LIN {X 0,Y 283.836,Z 555.722,A -85,B 0,C 180,E1 20309.781,E2 20309.781} C_VEL
LIN {X 0,Y 281.486,Z 550.799,A -85,B 0,C 180,E1 20310.705,E2 20310.705} C_VEL
LIN {X 0,Y 279.401,Z 540.674,A -85,B 0,C 180,E1 20314.395,E2 20314.395} C_VEL
LIN {X 0,Y 277.114,Z 531.716,A -85,B 0,C 180,E1 20318.183,E2 20318.183} C_VEL
LIN {X 0,Y 274.511,Z 522.89,A -85,B 0,C 180,E1 20322.608,E2 20322.608} C_VEL
LIN {X 0,Y 272.161,Z 516.128,A -85,B 0,C 180,E1 20326.833,E2 20326.833} C_VEL
LIN {X 0,Y 270.651,Z 512.243,A -85,B 0,C 180,E1 20329.786,E2 20329.786} C_VEL
LIN {X 0,Y 269.541,Z 509.144,A -85,B 0,C 180,E1 20332.54,E2 20332.54} C_VEL
LIN {X 0,Y 268.278,Z 505.702,A -85,B 0,C 180,E1 20336.367,E2 20336.367} C_VEL
LIN {X 0,Y 267.046,Z 502.186,A -85,B 0,C 180,E1 20343.219,E2 20343.219} C_VEL
LIN {X 0,Y 266.89,Z 501.903,A -85,B 0,C 180,E1 20348.618,E2 20348.618} C_VEL
LIN {X 0,Y 267.553,Z 502.917,A -85,B 0,C 180,E1 20352.744,E2 20352.744} C_VEL
LIN {X 0,Y 269.686,Z 507.312,A -85,B 0,C 180,E1 20359.492,E2 20359.492} C_VEL
LIN {X 0,Y 271.699,Z 511.865,A -85,B 0,C 180,E1 20363.648,E2 20363.648} C_VEL
LIN {X 0,Y 273.683,Z 516.523,A -85,B 0,C 180,E1 20366.949,E2 20366.949} C_VEL
LIN {X 0,Y 276.357,Z 522.601,A -85,B 0,C 180,E1 20370.562,E2 20370.562} C_VEL
LIN {X 0,Y 279.81,Z 531.752,A -85,B 0,C 180,E1 20374.871,E2 20374.871} C_VEL
LIN {X 0,Y 283.199,Z 541.616,A -85,B 0,C 180,E1 20378.676,E2 20378.676} C_VEL
LIN {X 0,Y 284.32,Z 544.973,A -85,B 0,C 180,E1 20379.794,E2 20379.794} C_VEL
LIN {X 0,Y 291.359,Z 556.974,A -85,B 0,C 180,E1 20382.037,E2 20382.037} C_VEL
LIN {X 0,Y 293.853,Z 561.883,A -85,B 0,C 180,E1 20382.784,E2 20382.784} C_VEL
LIN {X 0,Y 295.222,Z 584.167,A -85,B 0,C 180,E1 20383.897,E2 20383.897} C_VEL
LIN {X 0,Y 287.499,Z 725.367,A -85,B 0,C 180,E1 20387.325,E2 20387.325} C_VEL
LIN {X 0,Y 285.33,Z 743.573,A -85,B 0,C 180,E1 20388.063,E2 20388.063} C_VEL
LIN {X 0,Y 282.159,Z 761.285,A -85,B 0,C 180,E1 20389.11,E2 20389.11} C_VEL
LIN {X 0,Y 278.499,Z 777.354,A -85,B 0,C 180,E1 20390.413,E2 20390.413} C_VEL
LIN {X 0,Y 274.274,Z 793.21,A -85,B 0,C 180,E1 20392.102,E2 20392.102} C_VEL
LIN {X 0,Y 269.76,Z 808.181,A -85,B 0,C 180,E1 20394.153,E2 20394.153} C_VEL
LIN {X 0,Y 264.96,Z 822.734,A -85,B 0,C 180,E1 20396.698,E2 20396.698} C_VEL
LIN {X 0,Y 260.466,Z 835.727,A -85,B 0,C 180,E1 20399.555,E2 20399.555} C_VEL
LIN {X 0,Y 256.384,Z 847.663,A -85,B 0,C 180,E1 20402.853,E2 20402.853} C_VEL
LIN {X 0,Y 253.012,Z 858.122,A -85,B 0,C 180,E1 20406.476,E2 20406.476} C_VEL
LIN {X 0,Y 250.58,Z 867.042,A -85,B 0,C 180,E1 20410.417,E2 20410.417} C_VEL
LIN {X 0,Y 249.191,Z 874.327,A -85,B 0,C 180,E1 20414.644,E2 20414.644} C_VEL
LIN {X 0,Y 248.918,Z 879.669,A -85,B 0,C 180,E1 20418.884,E2 20418.884} C_VEL
LIN {X 0,Y 249.44,Z 883.153,A -85,B 0,C 180,E1 20423.094,E2 20423.094} C_VEL
LIN {X 0,Y 250.202,Z 884.696,A -85,B 0,C 180,E1 20426.793,E2 20426.793} C_VEL
LIN {X 0,Y 250.573,Z 884.807,A -85,B 0,C 180,E1 20430,E2 20430} C_VEL
LIN {X 0,Y 250.353,Z 883.594,A -85,B 0,C 180,E1 20433.206,E2 20433.206} C_VEL
LIN {X 0,Y 249.71,Z 880.685,A -85,B 0,C 180,E1 20436.9,E2 20436.9} C_VEL
LIN {X 0,Y 249.251,Z 876.121,A -85,B 0,C 180,E1 20440.641,E2 20440.641} C_VEL
LIN {X 0,Y 249.336,Z 869.417,A -85,B 0,C 180,E1 20444.634,E2 20444.634} C_VEL
LIN {X 0,Y 250.208,Z 861.167,A -85,B 0,C 180,E1 20448.403,E2 20448.403} C_VEL
LIN {X 0,Y 251.809,Z 851.451,A -85,B 0,C 180,E1 20451.916,E2 20451.916} C_VEL
LIN {X 0,Y 254.087,Z 840.281,A -85,B 0,C 180,E1 20455.168,E2 20455.168} C_VEL
LIN {X 0,Y 256.938,Z 827.315,A -85,B 0,C 180,E1 20458.217,E2 20458.217} C_VEL
LIN {X 0,Y 260.267,Z 812.638,A -85,B 0,C 180,E1 20460.983,E2 20460.983} C_VEL
LIN {X 0,Y 263.513,Z 797.555,A -85,B 0,C 180,E1 20463.25,E2 20463.25} C_VEL
LIN {X 0,Y 266.665,Z 781.594,A -85,B 0,C 180,E1 20465.139,E2 20465.139} C_VEL
LIN {X 0,Y 269.568,Z 764.639,A -85,B 0,C 180,E1 20466.668,E2 20466.668} C_VEL
LIN {X 0,Y 272.01,Z 746.93,A -85,B 0,C 180,E1 20467.836,E2 20467.836} C_VEL
LIN {X 0,Y 273.717,Z 728.333,A -85,B 0,C 180,E1 20468.673,E2 20468.673} C_VEL
LIN {X 0,Y 275.2,Z 692.013,A -85,B 0,C 180,E1 20469.616,E2 20469.616} C_VEL
LIN {X 0,Y 279.573,Z 578.588,A -85,B 0,C 180,E1 20472.411,E2 20472.411} C_VEL
LIN {X 0,Y 276.925,Z 544.256,A -85,B 0,C 180,E1 20473.808,E2 20473.808} C_VEL
LIN {X 0,Y 275.779,Z 540.484,A -85,B 0,C 180,E1 20474.568,E2 20474.568} C_VEL
LIN {X 0,Y 270.983,Z 524.24,A -85,B 0,C 180,E1 20478.506,E2 20478.506} C_VEL
LIN {X 0,Y 266.131,Z 509.628,A -85,B 0,C 180,E1 20482.509,E2 20482.509} C_VEL
LIN {X 0,Y 261.289,Z 496.731,A -85,B 0,C 180,E1 20486.562,E2 20486.562} C_VEL
LIN {X 0,Y 257.296,Z 486.923,A -85,B 0,C 180,E1 20490.065,E2 20490.065} C_VEL
LIN {X 0,Y 253.737,Z 478.944,A -85,B 0,C 180,E1 20493.307,E2 20493.307} C_VEL
LIN {X 0,Y 251.871,Z 474.922,A -85,B 0,C 180,E1 20495.116,E2 20495.116} C_VEL
LIN {X 0,Y 250.659,Z 471.661,A -85,B 0,C 180,E1 20496.74,E2 20496.74} C_VEL
LIN {X 0,Y 250.658,Z 471.575,A -85,B 0,C 180,E1 20501.691,E2 20501.691} C_VEL
LIN {X 0,Y 250.644,Z 471.547,A -85,B 0,C 180,E1 20506.623,E2 20506.623} C_VEL
LIN {X 0,Y 250.646,Z 471.525,A -85,B 0,C 180,E1 20511.744,E2 20511.744} C_VEL
LIN {X 0,Y 250.643,Z 471.573,A -85,B 0,C 180,E1 20516.57,E2 20516.57} C_VEL
LIN {X 0,Y 250.628,Z 471.528,A -85,B 0,C 180,E1 20521.601,E2 20521.601} C_VEL
LIN {X 0,Y 250.652,Z 471.536,A -85,B 0,C 180,E1 20526.413,E2 20526.413} C_VEL
LIN {X 0,Y 250.623,Z 471.552,A -85,B 0,C 180,E1 20531.507,E2 20531.507} C_VEL
LIN {X 0,Y 250.64,Z 471.519,A -85,B 0,C 180,E1 20536.454,E2 20536.454} C_VEL
LIN {X 0,Y 250.621,Z 471.578,A -85,B 0,C 180,E1 20541.534,E2 20541.534} C_VEL
LIN {X 0,Y 250.628,Z 471.52,A -85,B 0,C 180,E1 20546.54,E2 20546.54} C_VEL
LIN {X 0,Y 250.619,Z 471.565,A -85,B 0,C 180,E1 20551.375,E2 20551.375} C_VEL
LIN {X 0,Y 250.617,Z 471.551,A -85,B 0,C 180,E1 20556.474,E2 20556.474} C_VEL
LIN {X 0,Y 250.627,Z 471.535,A -85,B 0,C 180,E1 20561.168,E2 20561.168} C_VEL
LIN {X 0,Y 250.604,Z 471.553,A -85,B 0,C 180,E1 20566.351,E2 20566.351} C_VEL
LIN {X 0,Y 250.673,Z 471.876,A -85,B 0,C 180,E1 20569.265,E2 20569.265} C_VEL
LIN {X 0,Y 254.03,Z 480.157,A -85,B 0,C 180,E1 20573.253,E2 20573.253} C_VEL
LIN {X 0,Y 257.814,Z 489.79,A -85,B 0,C 180,E1 20577.379,E2 20577.379} C_VEL
LIN {X 0,Y 261.612,Z 500.82,A -85,B 0,C 180,E1 20581.528,E2 20581.528} C_VEL
LIN {X 0,Y 265.162,Z 512.595,A -85,B 0,C 180,E1 20585.494,E2 20585.494} C_VEL
LIN {X 0,Y 268.714,Z 526.333,A -85,B 0,C 180,E1 20589.665,E2 20589.665} C_VEL
LIN {X 0,Y 271.087,Z 537.756,A -85,B 0,C 180,E1 20592.838,E2 20592.838} C_VEL
LIN {X 0,Y 268.088,Z 551.998,A -85,B 0,C 180,E1 20595.687,E2 20595.687} C_VEL
LIN {X 0,Y 274.857,Z 601.391,A -85,B 0,C 180,E1 20598.171,E2 20598.171} C_VEL
LIN {X 0,Y 271.074,Z 689.431,A -85,B 0,C 180,E1 20600.552,E2 20600.552} C_VEL
LIN {X 0,Y 269.826,Z 706.849,A -85,B 0,C 180,E1 20601.442,E2 20601.442} C_VEL
LIN {X 0,Y 268.134,Z 722.124,A -85,B 0,C 180,E1 20602.608,E2 20602.608} C_VEL
LIN {X 0,Y 265.935,Z 737.206,A -85,B 0,C 180,E1 20604.173,E2 20604.173} C_VEL
LIN {X 0,Y 263.634,Z 750.147,A -85,B 0,C 180,E1 20605.921,E2 20605.921} C_VEL
LIN {X 0,Y 260.915,Z 763.556,A -85,B 0,C 180,E1 20608.243,E2 20608.243} C_VEL
LIN {X 0,Y 258.454,Z 774.558,A -85,B 0,C 180,E1 20610.665,E2 20610.665} C_VEL
LIN {X 0,Y 255.988,Z 784.977,A -85,B 0,C 180,E1 20613.583,E2 20613.583} C_VEL
LIN {X 0,Y 254.021,Z 793.252,A -85,B 0,C 180,E1 20616.554,E2 20616.554} C_VEL
LIN {X 0,Y 252.342,Z 800.574,A -85,B 0,C 180,E1 20620.04,E2 20620.04} C_VEL
LIN {X 0,Y 251.293,Z 805.904,A -85,B 0,C 180,E1 20623.577,E2 20623.577} C_VEL
LIN {X 0,Y 250.805,Z 809.6,A -85,B 0,C 180,E1 20627.397,E2 20627.397} C_VEL
LIN {X 0,Y 250.896,Z 811.325,A -85,B 0,C 180,E1 20631.018,E2 20631.018} C_VEL
LIN {X 0,Y 251.648,Z 811.302,A -85,B 0,C 180,E1 20635.054,E2 20635.054} C_VEL
LIN {X 0,Y 252.999,Z 809.49,A -85,B 0,C 180,E1 20638.674,E2 20638.674} C_VEL
LIN {X 0,Y 255.22,Z 805.65,A -85,B 0,C 180,E1 20642.46,E2 20642.46} C_VEL
LIN {X 0,Y 256.912,Z 802.391,A -85,B 0,C 180,E1 20644.646,E2 20644.646} C_VEL
LIN {X 0,Y 257.391,Z 799.759,A -85,B 0,C 180,E1 20646.272,E2 20646.272} C_VEL
LIN {X 0,Y 256.015,Z 793.806,A -85,B 0,C 180,E1 20649.761,E2 20649.761} C_VEL
LIN {X 0,Y 256.435,Z 789.726,A -85,B 0,C 180,E1 20651.519,E2 20651.519} C_VEL
LIN {X 0,Y 256.885,Z 788.523,A -85,B 0,C 180,E1 20651.925,E2 20651.925} C_VEL
LIN {X 0,Y 261.136,Z 778.548,A -85,B 0,C 180,E1 20654.79,E2 20654.79} C_VEL
LIN {X 0,Y 265.374,Z 767.255,A -85,B 0,C 180,E1 20657.282,E2 20657.282} C_VEL
LIN {X 0,Y 269.62,Z 754.388,A -85,B 0,C 180,E1 20659.483,E2 20659.483} C_VEL
LIN {X 0,Y 273.389,Z 740.659,A -85,B 0,C 180,E1 20661.288,E2 20661.288} C_VEL
LIN {X 0,Y 276.743,Z 725.457,A -85,B 0,C 180,E1 20662.811,E2 20662.811} C_VEL
LIN {X 0,Y 279.266,Z 709.934,A -85,B 0,C 180,E1 20663.947,E2 20663.947} C_VEL
LIN {X 0,Y 281.064,Z 693.204,A -85,B 0,C 180,E1 20664.784,E2 20664.784} C_VEL
LIN {X 0,Y 284.552,Z 637.632,A -85,B 0,C 180,E1 20666.321,E2 20666.321} C_VEL
LIN {X 0,Y 286.34,Z 606.894,A -85,B 0,C 180,E1 20667.127,E2 20667.127} C_VEL
LIN {X 0,Y 282.57,Z 579.868,A -85,B 0,C 180,E1 20669.101,E2 20669.101} C_VEL
LIN {X 0,Y 279.201,Z 560.292,A -85,B 0,C 180,E1 20670.795,E2 20670.795} C_VEL
LIN {X 0,Y 274.369,Z 550.897,A -85,B 0,C 180,E1 20672.666,E2 20672.666} C_VEL
LIN {X 0,Y 272.228,Z 541.418,A -85,B 0,C 180,E1 20676.4,E2 20676.4} C_VEL
LIN {X 0,Y 270.061,Z 533.036,A -85,B 0,C 180,E1 20680.311,E2 20680.311} C_VEL
LIN {X 0,Y 267.879,Z 525.784,A -85,B 0,C 180,E1 20684.361,E2 20684.361} C_VEL
LIN {X 0,Y 266.089,Z 520.654,A -85,B 0,C 180,E1 20687.852,E2 20687.852} C_VEL
LIN {X 0,Y 264.952,Z 517.461,A -85,B 0,C 180,E1 20690.442,E2 20690.442} C_VEL
LIN {X 0,Y 264.174,Z 515.07,A -85,B 0,C 180,E1 20692.606,E2 20692.606} C_VEL
LIN {X 0,Y 262.981,Z 511.675,A -85,B 0,C 180,E1 20696.512,E2 20696.512} C_VEL
LIN {X 0,Y 261.896,Z 508.303,A -85,B 0,C 180,E1 20703.283,E2 20703.283} C_VEL
LIN {X 0,Y 261.784,Z 508.061,A -85,B 0,C 180,E1 20708.566,E2 20708.566} C_VEL
LIN {X 0,Y 262.406,Z 508.985,A -85,B 0,C 180,E1 20712.544,E2 20712.544} C_VEL
LIN {X 0,Y 264.506,Z 513.468,A -85,B 0,C 180,E1 20719.429,E2 20719.429} C_VEL
LIN {X 0,Y 266.374,Z 517.771,A -85,B 0,C 180,E1 20723.445,E2 20723.445} C_VEL
LIN {X 0,Y 268.308,Z 522.441,A -85,B 0,C 180,E1 20726.802,E2 20726.802} C_VEL
LIN {X 0,Y 270.817,Z 528.375,A -85,B 0,C 180,E1 20730.384,E2 20730.384} C_VEL
LIN {X 0,Y 274.136,Z 537.344,A -85,B 0,C 180,E1 20734.679,E2 20734.679} C_VEL
LIN {X 0,Y 276.981,Z 545.541,A -85,B 0,C 180,E1 20737.855,E2 20737.855} C_VEL
LIN {X 0,Y 284.326,Z 557.623,A -85,B 0,C 180,E1 20740.386,E2 20740.386} C_VEL
LIN {X 0,Y 288.733,Z 565.802,A -85,B 0,C 180,E1 20741.772,E2 20741.772} C_VEL
LIN {X 0,Y 289.772,Z 585.519,A -85,B 0,C 180,E1 20742.765,E2 20742.765} C_VEL
LIN {X 0,Y 281.791,Z 724.625,A -85,B 0,C 180,E1 20746.184,E2 20746.184} C_VEL
LIN {X 0,Y 279.543,Z 742.778,A -85,B 0,C 180,E1 20746.927,E2 20746.927} C_VEL
LIN {X 0,Y 276.286,Z 760.314,A -85,B 0,C 180,E1 20747.972,E2 20747.972} C_VEL
LIN {X 0,Y 272.338,Z 776.921,A -85,B 0,C 180,E1 20749.333,E2 20749.333} C_VEL
LIN {X 0,Y 268.015,Z 792.409,A -85,B 0,C 180,E1 20751.006,E2 20751.006} C_VEL
LIN {X 0,Y 263.214,Z 807.553,A -85,B 0,C 180,E1 20753.117,E2 20753.117} C_VEL
LIN {X 0,Y 258.234,Z 821.902,A -85,B 0,C 180,E1 20755.676,E2 20755.676} C_VEL
LIN {X 0,Y 253.438,Z 834.976,A -85,B 0,C 180,E1 20758.617,E2 20758.617} C_VEL
LIN {X 0,Y 249.058,Z 846.981,A -85,B 0,C 180,E1 20762.031,E2 20762.031} C_VEL
LIN {X 0,Y 245.492,Z 857.227,A -85,B 0,C 180,E1 20765.71,E2 20765.71} C_VEL
LIN {X 0,Y 242.793,Z 866.249,A -85,B 0,C 180,E1 20769.874,E2 20769.874} C_VEL
LIN {X 0,Y 241.297,Z 873.292,A -85,B 0,C 180,E1 20774.129,E2 20774.129} C_VEL
LIN {X 0,Y 240.932,Z 878.589,A -85,B 0,C 180,E1 20778.51,E2 20778.51} C_VEL
LIN {X 0,Y 241.442,Z 882.03,A -85,B 0,C 180,E1 20782.864,E2 20782.864} C_VEL
LIN {X 0,Y 242.253,Z 883.527,A -85,B 0,C 180,E1 20786.688,E2 20786.688} C_VEL
LIN {X 0,Y 242.667,Z 883.582,A -85,B 0,C 180,E1 20790,E2 20790} C_VEL
LIN {X 0,Y 242.418,Z 882.329,A -85,B 0,C 180,E1 20793.311,E2 20793.311} C_VEL
LIN {X 0,Y 241.756,Z 879.472,A -85,B 0,C 180,E1 20796.978,E2 20796.978} C_VEL
LIN {X 0,Y 241.277,Z 874.675,A -85,B 0,C 180,E1 20800.99,E2 20800.99} C_VEL
LIN {X 0,Y 241.425,Z 867.852,A -85,B 0,C 180,E1 20805.125,E2 20805.125} C_VEL
LIN {X 0,Y 242.416,Z 859.446,A -85,B 0,C 180,E1 20809.017,E2 20809.017} C_VEL
LIN {X 0,Y 244.172,Z 849.557,A -85,B 0,C 180,E1 20812.639,E2 20812.639} C_VEL
LIN {X 0,Y 246.612,Z 838.276,A -85,B 0,C 180,E1 20815.969,E2 20815.969} C_VEL
LIN {X 0,Y 249.675,Z 825.042,A -85,B 0,C 180,E1 20819.116,E2 20819.116} C_VEL
LIN {X 0,Y 253.093,Z 810.625,A -85,B 0,C 180,E1 20821.857,E2 20821.857} C_VEL
LIN {X 0,Y 256.467,Z 795.449,A -85,B 0,C 180,E1 20824.153,E2 20824.153} C_VEL
LIN {X 0,Y 259.775,Z 779.069,A -85,B 0,C 180,E1 20826.079,E2 20826.079} C_VEL
LIN {X 0,Y 262.694,Z 762.248,A -85,B 0,C 180,E1 20827.586,E2 20827.586} C_VEL
LIN {X 0,Y 265.223,Z 744.034,A -85,B 0,C 180,E1 20828.767,E2 20828.767} C_VEL
LIN {X 0,Y 266.838,Z 725.763,A -85,B 0,C 180,E1 20829.569,E2 20829.569} C_VEL
LIN {X 0,Y 272.749,Z 579.371,A -85,B 0,C 180,E1 20833.27,E2 20833.27} C_VEL
LIN {X 0,Y 270.362,Z 547.278,A -85,B 0,C 180,E1 20834.61,E2 20834.61} C_VEL
LIN {X 0,Y 268.705,Z 543.649,A -85,B 0,C 180,E1 20835.009,E2 20835.009} C_VEL
LIN {X 0,Y 263.955,Z 527.386,A -85,B 0,C 180,E1 20839.056,E2 20839.056} C_VEL
LIN {X 0,Y 259.337,Z 513.333,A -85,B 0,C 180,E1 20843.027,E2 20843.027} C_VEL
LIN {X 0,Y 254.872,Z 501.19,A -85,B 0,C 180,E1 20846.956,E2 20846.956} C_VEL
LIN {X 0,Y 251.089,Z 491.766,A -85,B 0,C 180,E1 20850.411,E2 20850.411} C_VEL
LIN {X 0,Y 247.7,Z 483.997,A -85,B 0,C 180,E1 20853.653,E2 20853.653} C_VEL
LIN {X 0,Y 245.836,Z 479.986,A -85,B 0,C 180,E1 20855.49,E2 20855.49} C_VEL
LIN {X 0,Y 244.092,Z 476.123,A -85,B 0,C 180,E1 20857.354,E2 20857.354} C_VEL
LIN {X 0,Y 242.724,Z 472.655,A -85,B 0,C 180,E1 20859.252,E2 20859.252} C_VEL
LIN {X 0,Y 242.713,Z 472.52,A -85,B 0,C 180,E1 20864.224,E2 20864.224} C_VEL
LIN {X 0,Y 242.699,Z 472.547,A -85,B 0,C 180,E1 20869.317,E2 20869.317} C_VEL
LIN {X 0,Y 242.712,Z 472.535,A -85,B 0,C 180,E1 20874.326,E2 20874.326} C_VEL
LIN {X 0,Y 242.689,Z 472.507,A -85,B 0,C 180,E1 20879.528,E2 20879.528} C_VEL
LIN {X 0,Y 242.706,Z 472.563,A -85,B 0,C 180,E1 20884.49,E2 20884.49} C_VEL
LIN {X 0,Y 242.682,Z 472.505,A -85,B 0,C 180,E1 20889.486,E2 20889.486} C_VEL
LIN {X 0,Y 242.717,Z 472.54,A -85,B 0,C 180,E1 20894.554,E2 20894.554} C_VEL
LIN {X 0,Y 242.68,Z 472.525,A -85,B 0,C 180,E1 20899.746,E2 20899.746} C_VEL
LIN {X 0,Y 242.694,Z 472.518,A -85,B 0,C 180,E1 20904.589,E2 20904.589} C_VEL
LIN {X 0,Y 242.676,Z 472.562,A -85,B 0,C 180,E1 20909.632,E2 20909.632} C_VEL
LIN {X 0,Y 242.681,Z 472.516,A -85,B 0,C 180,E1 20914.651,E2 20914.651} C_VEL
LIN {X 0,Y 242.669,Z 472.538,A -85,B 0,C 180,E1 20919.691,E2 20919.691} C_VEL
LIN {X 0,Y 242.683,Z 472.567,A -85,B 0,C 180,E1 20924.875,E2 20924.875} C_VEL
LIN {X 0,Y 242.718,Z 472.845,A -85,B 0,C 180,E1 20926.752,E2 20926.752} C_VEL
LIN {X 0,Y 244.736,Z 477.914,A -85,B 0,C 180,E1 20929.489,E2 20929.489} C_VEL
LIN {X 0,Y 246.68,Z 482.601,A -85,B 0,C 180,E1 20931.845,E2 20931.845} C_VEL
LIN {X 0,Y 249.322,Z 489.202,A -85,B 0,C 180,E1 20934.896,E2 20934.896} C_VEL
LIN {X 0,Y 252.512,Z 497.795,A -85,B 0,C 180,E1 20938.488,E2 20938.488} C_VEL
LIN {X 0,Y 256.337,Z 509.545,A -85,B 0,C 180,E1 20942.847,E2 20942.847} C_VEL
LIN {X 0,Y 259.74,Z 521.916,A -85,B 0,C 180,E1 20946.931,E2 20946.931} C_VEL
LIN {X 0,Y 262.951,Z 535.608,A -85,B 0,C 180,E1 20951.027,E2 20951.027} C_VEL
LIN {X 0,Y 263.739,Z 540.393,A -85,B 0,C 180,E1 20952.344,E2 20952.344} C_VEL
LIN {X 0,Y 261.246,Z 551.57,A -85,B 0,C 180,E1 20954.636,E2 20954.636} C_VEL
LIN {X 0,Y 268.01,Z 602.213,A -85,B 0,C 180,E1 20957.305,E2 20957.305} C_VEL
LIN {X 0,Y 264.079,Z 690.008,A -85,B 0,C 180,E1 20959.728,E2 20959.728} C_VEL
LIN {X 0,Y 262.777,Z 707.452,A -85,B 0,C 180,E1 20960.638,E2 20960.638} C_VEL
LIN {X 0,Y 260.984,Z 722.984,A -85,B 0,C 180,E1 20961.85,E2 20961.85} C_VEL
LIN {X 0,Y 258.628,Z 738.466,A -85,B 0,C 180,E1 20963.501,E2 20963.501} C_VEL
LIN {X 0,Y 256.084,Z 752.036,A -85,B 0,C 180,E1 20965.409,E2 20965.409} C_VEL
LIN {X 0,Y 253.338,Z 764.997,A -85,B 0,C 180,E1 20967.738,E2 20967.738} C_VEL
LIN {X 0,Y 250.782,Z 775.895,A -85,B 0,C 180,E1 20970.228,E2 20970.228} C_VEL
LIN {X 0,Y 248.224,Z 786.264,A -85,B 0,C 180,E1 20973.232,E2 20973.232} C_VEL
LIN {X 0,Y 246.181,Z 794.486,A -85,B 0,C 180,E1 20976.295,E2 20976.295} C_VEL
LIN {X 0,Y 244.444,Z 801.784,A -85,B 0,C 180,E1 20979.892,E2 20979.892} C_VEL
LIN {X 0,Y 243.364,Z 807.092,A -85,B 0,C 180,E1 20983.543,E2 20983.543} C_VEL
LIN {X 0,Y 242.875,Z 810.785,A -85,B 0,C 180,E1 20987.489,E2 20987.489} C_VEL
LIN {X 0,Y 242.998,Z 812.509,A -85,B 0,C 180,E1 20991.228,E2 20991.228} C_VEL
LIN {X 0,Y 243.783,Z 812.523,A -85,B 0,C 180,E1 20995.248,E2 20995.248} C_VEL
LIN {X 0,Y 245.24,Z 810.778,A -85,B 0,C 180,E1 20999.023,E2 20999.023} C_VEL
LIN {X 0,Y 247.532,Z 807.102,A -85,B 0,C 180,E1 21002.84,E2 21002.84} C_VEL
LIN {X 0,Y 250.35,Z 802.036,A -85,B 0,C 180,E1 21006.234,E2 21006.234} C_VEL
LIN {X 0,Y 253.953,Z 794.834,A -85,B 0,C 180,E1 21009.629,E2 21009.629} C_VEL
LIN {X 0,Y 256.885,Z 788.523,A -85,B 0,C 180,E1 21011.925,E2 21011.925} C_VEL
LIN {X 0,Y 257.925,Z 784.369,A -85,B 0,C 180,E1 21013.369,E2 21013.369} C_VEL
LIN {X 0,Y 257.733,Z 774.755,A -85,B 0,C 180,E1 21016.723,E2 21016.723} C_VEL
LIN {X 0,Y 258.551,Z 769.785,A -85,B 0,C 180,E1 21018.026,E2 21018.026} C_VEL
LIN {X 0,Y 259.064,Z 768.194,A -85,B 0,C 180,E1 21018.352,E2 21018.352} C_VEL
LIN {X 0,Y 263.465,Z 755.484,A -85,B 0,C 180,E1 21020.559,E2 21020.559} C_VEL
LIN {X 0,Y 267.236,Z 742.498,A -85,B 0,C 180,E1 21022.309,E2 21022.309} C_VEL
LIN {X 0,Y 270.659,Z 727.884,A -85,B 0,C 180,E1 21023.821,E2 21023.821} C_VEL
LIN {X 0,Y 273.445,Z 712.209,A -85,B 0,C 180,E1 21025.025,E2 21025.025} C_VEL
LIN {X 0,Y 275.401,Z 695.375,A -85,B 0,C 180,E1 21025.904,E2 21025.904} C_VEL
LIN {X 0,Y 277.342,Z 666.078,A -85,B 0,C 180,E1 21026.789,E2 21026.789} C_VEL
LIN {X 0,Y 280.993,Z 608.321,A -85,B 0,C 180,E1 21028.316,E2 21028.316} C_VEL
LIN {X 0,Y 277.513,Z 581.897,A -85,B 0,C 180,E1 21030.318,E2 21030.318} C_VEL
LIN {X 0,Y 274.693,Z 564.8,A -85,B 0,C 180,E1 21031.847,E2 21031.847} C_VEL
LIN {X 0,Y 269.136,Z 554.591,A -85,B 0,C 180,E1 21033.999,E2 21033.999} C_VEL
LIN {X 0,Y 266.987,Z 550.224,A -85,B 0,C 180,E1 21035.082,E2 21035.082} C_VEL
LIN {X 0,Y 264.977,Z 541.436,A -85,B 0,C 180,E1 21038.993,E2 21038.993} C_VEL
LIN {X 0,Y 262.865,Z 533.531,A -85,B 0,C 180,E1 21043.197,E2 21043.197} C_VEL
LIN {X 0,Y 260.837,Z 527.179,A -85,B 0,C 180,E1 21047.379,E2 21047.379} C_VEL
LIN {X 0,Y 259.503,Z 523.334,A -85,B 0,C 180,E1 21050.525,E2 21050.525} C_VEL
LIN {X 0,Y 258.693,Z 520.81,A -85,B 0,C 180,E1 21052.895,E2 21052.895} C_VEL
LIN {X 0,Y 257.681,Z 517.645,A -85,B 0,C 180,E1 21056.663,E2 21056.663} C_VEL
LIN {X 0,Y 256.746,Z 514.419,A -85,B 0,C 180,E1 21063.348,E2 21063.348} C_VEL
LIN {X 0,Y 256.704,Z 514.244,A -85,B 0,C 180,E1 21068.737,E2 21068.737} C_VEL
LIN {X 0,Y 257.297,Z 515.177,A -85,B 0,C 180,E1 21072.569,E2 21072.569} C_VEL
LIN {X 0,Y 259.244,Z 519.346,A -85,B 0,C 180,E1 21079.137,E2 21079.137} C_VEL
LIN {X 0,Y 261.044,Z 523.67,A -85,B 0,C 180,E1 21083.235,E2 21083.235} C_VEL
LIN {X 0,Y 262.926,Z 528.362,A -85,B 0,C 180,E1 21086.664,E2 21086.664} C_VEL
LIN {X 0,Y 265.222,Z 533.936,A -85,B 0,C 180,E1 21090.092,E2 21090.092} C_VEL
LIN {X 0,Y 268.443,Z 542.938,A -85,B 0,C 180,E1 21094.482,E2 21094.482} C_VEL
LIN {X 0,Y 269.683,Z 546.15,A -85,B 0,C 180,E1 21095.714,E2 21095.714} C_VEL
LIN {X 0,Y 277.429,Z 558.407,A -85,B 0,C 180,E1 21098.604,E2 21098.604} C_VEL
LIN {X 0,Y 283.681,Z 569.533,A -85,B 0,C 180,E1 21100.711,E2 21100.711} C_VEL
LIN {X 0,Y 284.453,Z 586.644,A -85,B 0,C 180,E1 21101.585,E2 21101.585} C_VEL
LIN {X 0,Y 276.223,Z 723.893,A -85,B 0,C 180,E1 21104.992,E2 21104.992} C_VEL
LIN {X 0,Y 273.912,Z 741.932,A -85,B 0,C 180,E1 21105.733,E2 21105.733} C_VEL
LIN {X 0,Y 270.661,Z 758.92,A -85,B 0,C 180,E1 21106.744,E2 21106.744} C_VEL
LIN {X 0,Y 266.551,Z 775.639,A -85,B 0,C 180,E1 21108.111,E2 21108.111} C_VEL
LIN {X 0,Y 261.943,Z 791.437,A -85,B 0,C 180,E1 21109.828,E2 21109.828} C_VEL
LIN {X 0,Y 257.023,Z 806.234,A -85,B 0,C 180,E1 21111.911,E2 21111.911} C_VEL
LIN {X 0,Y 251.688,Z 820.831,A -85,B 0,C 180,E1 21114.55,E2 21114.55} C_VEL
LIN {X 0,Y 246.484,Z 834.224,A -85,B 0,C 180,E1 21117.626,E2 21117.626} C_VEL
LIN {X 0,Y 241.881,Z 846.045,A -85,B 0,C 180,E1 21121.077,E2 21121.077} C_VEL
LIN {X 0,Y 238.017,Z 856.354,A -85,B 0,C 180,E1 21124.895,E2 21124.895} C_VEL
LIN {X 0,Y 235.142,Z 865.093,A -85,B 0,C 180,E1 21129.073,E2 21129.073} C_VEL
LIN {X 0,Y 233.419,Z 872.26,A -85,B 0,C 180,E1 21133.578,E2 21133.578} C_VEL
LIN {X 0,Y 232.951,Z 877.523,A -85,B 0,C 180,E1 21138.126,E2 21138.126} C_VEL
LIN {X 0,Y 233.439,Z 880.905,A -85,B 0,C 180,E1 21142.618,E2 21142.618} C_VEL
LIN {X 0,Y 234.303,Z 882.358,A -85,B 0,C 180,E1 21146.575,E2 21146.575} C_VEL
LIN {X 0,Y 234.761,Z 882.355,A -85,B 0,C 180,E1 21150,E2 21150} C_VEL
LIN {X 0,Y 234.479,Z 881.062,A -85,B 0,C 180,E1 21153.423,E2 21153.423} C_VEL
LIN {X 0,Y 233.744,Z 877.971,A -85,B 0,C 180,E1 21157.373,E2 21157.373} C_VEL
LIN {X 0,Y 233.289,Z 872.879,A -85,B 0,C 180,E1 21161.622,E2 21161.622} C_VEL
LIN {X 0,Y 233.574,Z 865.766,A -85,B 0,C 180,E1 21165.901,E2 21165.901} C_VEL
LIN {X 0,Y 234.746,Z 857.081,A -85,B 0,C 180,E1 21169.923,E2 21169.923} C_VEL
LIN {X 0,Y 236.74,Z 846.916,A -85,B 0,C 180,E1 21173.655,E2 21173.655} C_VEL
LIN {X 0,Y 239.424,Z 835.313,A -85,B 0,C 180,E1 21177.078,E2 21177.078} C_VEL
LIN {X 0,Y 242.616,Z 822.205,A -85,B 0,C 180,E1 21180.185,E2 21180.185} C_VEL
LIN {X 0,Y 246.07,Z 808.109,A -85,B 0,C 180,E1 21182.851,E2 21182.851} C_VEL
LIN {X 0,Y 249.492,Z 793.12,A -85,B 0,C 180,E1 21185.106,E2 21185.106} C_VEL
LIN {X 0,Y 252.756,Z 777.412,A -85,B 0,C 180,E1 21186.962,E2 21186.962} C_VEL
LIN {X 0,Y 255.895,Z 759.678,A -85,B 0,C 180,E1 21188.552,E2 21188.552} C_VEL
LIN {X 0,Y 258.387,Z 741.833,A -85,B 0,C 180,E1 21189.698,E2 21189.698} C_VEL
LIN {X 0,Y 259.963,Z 723.515,A -85,B 0,C 180,E1 21190.482,E2 21190.482} C_VEL
LIN {X 0,Y 265.988,Z 580.2,A -85,B 0,C 180,E1 21194.171,E2 21194.171} C_VEL
LIN {X 0,Y 263.773,Z 550.145,A -85,B 0,C 180,E1 21195.472,E2 21195.472} C_VEL
LIN {X 0,Y 260.762,Z 543.756,A -85,B 0,C 180,E1 21196.204,E2 21196.204} C_VEL
LIN {X 0,Y 256.253,Z 528.312,A -85,B 0,C 180,E1 21200.235,E2 21200.235} C_VEL
LIN {X 0,Y 251.793,Z 514.778,A -85,B 0,C 180,E1 21204.287,E2 21204.287} C_VEL
LIN {X 0,Y 247.708,Z 503.625,A -85,B 0,C 180,E1 21208.078,E2 21208.078} C_VEL
LIN {X 0,Y 243.568,Z 493.357,A -85,B 0,C 180,E1 21212.097,E2 21212.097} C_VEL
LIN {X 0,Y 240.074,Z 485.499,A -85,B 0,C 180,E1 21215.65,E2 21215.65} C_VEL
LIN {X 0,Y 238.101,Z 481.221,A -85,B 0,C 180,E1 21217.794,E2 21217.794} C_VEL
LIN {X 0,Y 236.265,Z 477.26,A -85,B 0,C 180,E1 21219.954,E2 21219.954} C_VEL
LIN {X 0,Y 234.791,Z 473.639,A -85,B 0,C 180,E1 21222.145,E2 21222.145} C_VEL
LIN {X 0,Y 234.763,Z 473.534,A -85,B 0,C 180,E1 21227.245,E2 21227.245} C_VEL
LIN {X 0,Y 234.768,Z 473.5,A -85,B 0,C 180,E1 21232.414,E2 21232.414} C_VEL
LIN {X 0,Y 234.756,Z 473.522,A -85,B 0,C 180,E1 21237.559,E2 21237.559} C_VEL
LIN {X 0,Y 234.764,Z 473.515,A -85,B 0,C 180,E1 21242.441,E2 21242.441} C_VEL
LIN {X 0,Y 234.743,Z 473.495,A -85,B 0,C 180,E1 21247.588,E2 21247.588} C_VEL
LIN {X 0,Y 234.762,Z 473.552,A -85,B 0,C 180,E1 21252.754,E2 21252.754} C_VEL
LIN {X 0,Y 234.747,Z 473.491,A -85,B 0,C 180,E1 21258.116,E2 21258.116} C_VEL
LIN {X 0,Y 234.752,Z 473.538,A -85,B 0,C 180,E1 21263.074,E2 21263.074} C_VEL
LIN {X 0,Y 234.757,Z 473.517,A -85,B 0,C 180,E1 21268.492,E2 21268.492} C_VEL
LIN {X 0,Y 234.736,Z 473.506,A -85,B 0,C 180,E1 21273.397,E2 21273.397} C_VEL
LIN {X 0,Y 234.756,Z 473.54,A -85,B 0,C 180,E1 21278.791,E2 21278.791} C_VEL
LIN {X 0,Y 234.751,Z 473.719,A -85,B 0,C 180,E1 21283.797,E2 21283.797} C_VEL
LIN {X 0,Y 236.935,Z 479.069,A -85,B 0,C 180,E1 21287.069,E2 21287.069} C_VEL
LIN {X 0,Y 238.65,Z 483.101,A -85,B 0,C 180,E1 21289.318,E2 21289.318} C_VEL
LIN {X 0,Y 241.282,Z 489.217,A -85,B 0,C 180,E1 21292.471,E2 21292.471} C_VEL
LIN {X 0,Y 244.978,Z 499.252,A -85,B 0,C 180,E1 21296.97,E2 21296.97} C_VEL
LIN {X 0,Y 248.414,Z 509.772,A -85,B 0,C 180,E1 21301.118,E2 21301.118} C_VEL
LIN {X 0,Y 251.744,Z 521.447,A -85,B 0,C 180,E1 21305.227,E2 21305.227} C_VEL
LIN {X 0,Y 254.85,Z 534.36,A -85,B 0,C 180,E1 21309.323,E2 21309.323} C_VEL
LIN {X 0,Y 256.408,Z 543.022,A -85,B 0,C 180,E1 21311.822,E2 21311.822} C_VEL
LIN {X 0,Y 254.451,Z 551.786,A -85,B 0,C 180,E1 21313.616,E2 21313.616} C_VEL
LIN {X 0,Y 261.22,Z 603.224,A -85,B 0,C 180,E1 21316.398,E2 21316.398} C_VEL
LIN {X 0,Y 257.142,Z 690.584,A -85,B 0,C 180,E1 21318.86,E2 21318.86} C_VEL
LIN {X 0,Y 255.792,Z 707.95,A -85,B 0,C 180,E1 21319.783,E2 21319.783} C_VEL
LIN {X 0,Y 254.048,Z 722.704,A -85,B 0,C 180,E1 21320.942,E2 21320.942} C_VEL
LIN {X 0,Y 251.651,Z 737.992,A -85,B 0,C 180,E1 21322.58,E2 21322.58} C_VEL
LIN {X 0,Y 249.07,Z 751.516,A -85,B 0,C 180,E1 21324.471,E2 21324.471} C_VEL
LIN {X 0,Y 246.167,Z 764.721,A -85,B 0,C 180,E1 21326.856,E2 21326.856} C_VEL
LIN {X 0,Y 243.352,Z 776.346,A -85,B 0,C 180,E1 21329.529,E2 21329.529} C_VEL
LIN {X 0,Y 240.652,Z 786.817,A -85,B 0,C 180,E1 21332.619,E2 21332.619} C_VEL
LIN {X 0,Y 238.493,Z 795.171,A -85,B 0,C 180,E1 21335.774,E2 21335.774} C_VEL
LIN {X 0,Y 236.644,Z 802.563,A -85,B 0,C 180,E1 21339.484,E2 21339.484} C_VEL
LIN {X 0,Y 235.49,Z 807.999,A -85,B 0,C 180,E1 21343.254,E2 21343.254} C_VEL
LIN {X 0,Y 234.955,Z 811.786,A -85,B 0,C 180,E1 21347.33,E2 21347.33} C_VEL
LIN {X 0,Y 235.091,Z 813.672,A -85,B 0,C 180,E1 21351.34,E2 21351.34} C_VEL
LIN {X 0,Y 235.967,Z 813.717,A -85,B 0,C 180,E1 21355.607,E2 21355.607} C_VEL
LIN {X 0,Y 237.542,Z 811.987,A -85,B 0,C 180,E1 21359.503,E2 21359.503} C_VEL
LIN {X 0,Y 239.947,Z 808.406,A -85,B 0,C 180,E1 21363.37,E2 21363.37} C_VEL
LIN {X 0,Y 243.149,Z 803.022,A -85,B 0,C 180,E1 21367.083,E2 21367.083} C_VEL
LIN {X 0,Y 247.113,Z 795.584,A -85,B 0,C 180,E1 21370.649,E2 21370.649} C_VEL
LIN {X 0,Y 251.056,Z 787.517,A -85,B 0,C 180,E1 21373.55,E2 21373.55} C_VEL
LIN {X 0,Y 255.526,Z 777.234,A -85,B 0,C 180,E1 21376.376,E2 21376.376} C_VEL
LIN {X 0,Y 259.064,Z 768.194,A -85,B 0,C 180,E1 21378.352,E2 21378.352} C_VEL
LIN {X 0,Y 260.324,Z 762.708,A -85,B 0,C 180,E1 21379.534,E2 21379.534} C_VEL
LIN {X 0,Y 260.54,Z 750.247,A -85,B 0,C 180,E1 21382.358,E2 21382.358} C_VEL
LIN {X 0,Y 261.283,Z 744.143,A -85,B 0,C 180,E1 21383.385,E2 21383.385} C_VEL
LIN {X 0,Y 261.725,Z 742.236,A -85,B 0,C 180,E1 21383.622,E2 21383.622} C_VEL
LIN {X 0,Y 265.445,Z 726.766,A -85,B 0,C 180,E1 21385.199,E2 21385.199} C_VEL
LIN {X 0,Y 268.25,Z 710.802,A -85,B 0,C 180,E1 21386.378,E2 21386.378} C_VEL
LIN {X 0,Y 270.198,Z 694.114,A -85,B 0,C 180,E1 21387.22,E2 21387.22} C_VEL
LIN {X 0,Y 274.468,Z 631.564,A -85,B 0,C 180,E1 21388.961,E2 21388.961} C_VEL
LIN {X 0,Y 275.809,Z 609.719,A -85,B 0,C 180,E1 21389.56,E2 21389.56} C_VEL
LIN {X 0,Y 272.576,Z 583.8,A -85,B 0,C 180,E1 21391.593,E2 21391.593} C_VEL
LIN {X 0,Y 270.292,Z 569.258,A -85,B 0,C 180,E1 21392.935,E2 21392.935} C_VEL
LIN {X 0,Y 263.981,Z 557.548,A -85,B 0,C 180,E1 21395.556,E2 21395.556} C_VEL
LIN {X 0,Y 259.83,Z 550.123,A -85,B 0,C 180,E1 21397.606,E2 21397.606} C_VEL
LIN {X 0,Y 257.779,Z 541.6,A -85,B 0,C 180,E1 21401.922,E2 21401.922} C_VEL
LIN {X 0,Y 255.912,Z 535.077,A -85,B 0,C 180,E1 21405.981,E2 21405.981} C_VEL
LIN {X 0,Y 254.304,Z 529.816,A -85,B 0,C 180,E1 21410.037,E2 21410.037} C_VEL
LIN {X 0,Y 253.233,Z 526.558,A -85,B 0,C 180,E1 21413.197,E2 21413.197} C_VEL
LIN {X 0,Y 252.377,Z 523.609,A -85,B 0,C 180,E1 21416.82,E2 21416.82} C_VEL
LIN {X 0,Y 251.577,Z 520.52,A -85,B 0,C 180,E1 21423.417,E2 21423.417} C_VEL
LIN {X 0,Y 251.6,Z 520.407,A -85,B 0,C 180,E1 21428.916,E2 21428.916} C_VEL
LIN {X 0,Y 252.173,Z 521.358,A -85,B 0,C 180,E1 21432.595,E2 21432.595} C_VEL
LIN {X 0,Y 254.061,Z 525.592,A -85,B 0,C 180,E1 21439.176,E2 21439.176} C_VEL
LIN {X 0,Y 255.807,Z 529.886,A -85,B 0,C 180,E1 21443.251,E2 21443.251} C_VEL
LIN {X 0,Y 257.544,Z 534.273,A -85,B 0,C 180,E1 21446.517,E2 21446.517} C_VEL
LIN {X 0,Y 259.897,Z 540.409,A -85,B 0,C 180,E1 21450.263,E2 21450.263} C_VEL
LIN {X 0,Y 262.123,Z 546.249,A -85,B 0,C 180,E1 21453.121,E2 21453.121} C_VEL
LIN {X 0,Y 268.743,Z 556.331,A -85,B 0,C 180,E1 21455.938,E2 21455.938} C_VEL
LIN {X 0,Y 275.995,Z 568.325,A -85,B 0,C 180,E1 21458.643,E2 21458.643} C_VEL
LIN {X 0,Y 278.798,Z 573.912,A -85,B 0,C 180,E1 21459.645,E2 21459.645} C_VEL
LIN {X 0,Y 279.278,Z 587.877,A -85,B 0,C 180,E1 21460.358,E2 21460.358} C_VEL
LIN {X 0,Y 270.76,Z 723.325,A -85,B 0,C 180,E1 21463.757,E2 21463.757} C_VEL
LIN {X 0,Y 268.35,Z 741.415,A -85,B 0,C 180,E1 21464.507,E2 21464.507} C_VEL
LIN {X 0,Y 264.876,Z 758.816,A -85,B 0,C 180,E1 21465.555,E2 21465.555} C_VEL
LIN {X 0,Y 260.619,Z 775.376,A -85,B 0,C 180,E1 21466.93,E2 21466.93} C_VEL
LIN {X 0,Y 255.825,Z 791.045,A -85,B 0,C 180,E1 21468.661,E2 21468.661} C_VEL
LIN {X 0,Y 250.415,Z 806.424,A -85,B 0,C 180,E1 21470.887,E2 21470.887} C_VEL
LIN {X 0,Y 244.93,Z 820.621,A -85,B 0,C 180,E1 21473.532,E2 21473.532} C_VEL
LIN {X 0,Y 239.612,Z 833.489,A -85,B 0,C 180,E1 21476.578,E2 21476.578} C_VEL
LIN {X 0,Y 234.729,Z 845.236,A -85,B 0,C 180,E1 21480.108,E2 21480.108} C_VEL
LIN {X 0,Y 230.596,Z 855.466,A -85,B 0,C 180,E1 21484.028,E2 21484.028} C_VEL
LIN {X 0,Y 227.476,Z 864.14,A -85,B 0,C 180,E1 21488.333,E2 21488.333} C_VEL
LIN {X 0,Y 225.56,Z 871.253,A -85,B 0,C 180,E1 21492.989,E2 21492.989} C_VEL
LIN {X 0,Y 224.972,Z 876.434,A -85,B 0,C 180,E1 21497.683,E2 21497.683} C_VEL
LIN {X 0,Y 225.437,Z 879.78,A -85,B 0,C 180,E1 21502.354,E2 21502.354} C_VEL
LIN {X 0,Y 226.372,Z 881.209,A -85,B 0,C 180,E1 21506.571,E2 21506.571} C_VEL
LIN {X 0,Y 226.856,Z 881.128,A -85,B 0,C 180,E1 21510,E2 21510} C_VEL
LIN {X 0,Y 226.58,Z 879.915,A -85,B 0,C 180,E1 21513.289,E2 21513.289} C_VEL
LIN {X 0,Y 225.811,Z 876.885,A -85,B 0,C 180,E1 21517.326,E2 21517.326} C_VEL
LIN {X 0,Y 225.339,Z 872.091,A -85,B 0,C 180,E1 21521.518,E2 21521.518} C_VEL
LIN {X 0,Y 225.6,Z 865.134,A -85,B 0,C 180,E1 21525.95,E2 21525.95} C_VEL
LIN {X 0,Y 226.797,Z 856.549,A -85,B 0,C 180,E1 21530.113,E2 21530.113} C_VEL
LIN {X 0,Y 228.945,Z 846.073,A -85,B 0,C 180,E1 21534.112,E2 21534.112} C_VEL
LIN {X 0,Y 231.853,Z 834.069,A -85,B 0,C 180,E1 21537.759,E2 21537.759} C_VEL
LIN {X 0,Y 235.215,Z 820.912,A -85,B 0,C 180,E1 21540.955,E2 21540.955} C_VEL
LIN {X 0,Y 238.823,Z 806.709,A -85,B 0,C 180,E1 21543.692,E2 21543.692} C_VEL
LIN {X 0,Y 242.402,Z 791.617,A -85,B 0,C 180,E1 21546,E2 21546} C_VEL
LIN {X 0,Y 246.008,Z 774.701,A -85,B 0,C 180,E1 21548.007,E2 21548.007} C_VEL
LIN {X 0,Y 249.069,Z 757.785,A -85,B 0,C 180,E1 21549.516,E2 21549.516} C_VEL
LIN {X 0,Y 251.59,Z 739.806,A -85,B 0,C 180,E1 21550.665,E2 21550.665} C_VEL
LIN {X 0,Y 253.13,Z 721.417,A -85,B 0,C 180,E1 21551.434,E2 21551.434} C_VEL
LIN {X 0,Y 259.285,Z 580.853,A -85,B 0,C 180,E1 21555.126,E2 21555.126} C_VEL
LIN {X 0,Y 257.342,Z 553.112,A -85,B 0,C 180,E1 21556.36,E2 21556.36} C_VEL
LIN {X 0,Y 252.877,Z 543.877,A -85,B 0,C 180,E1 21557.459,E2 21557.459} C_VEL
LIN {X 0,Y 248.646,Z 529.44,A -85,B 0,C 180,E1 21561.444,E2 21561.444} C_VEL
LIN {X 0,Y 244.548,Z 516.982,A -85,B 0,C 180,E1 21565.368,E2 21565.368} C_VEL
LIN {X 0,Y 240.086,Z 504.882,A -85,B 0,C 180,E1 21569.741,E2 21569.741} C_VEL
LIN {X 0,Y 236.13,Z 495.068,A -85,B 0,C 180,E1 21573.873,E2 21573.873} C_VEL
LIN {X 0,Y 232.603,Z 487.121,A -85,B 0,C 180,E1 21577.774,E2 21577.774} C_VEL
LIN {X 0,Y 230.455,Z 482.646,A -85,B 0,C 180,E1 21580.303,E2 21580.303} C_VEL
LIN {X 0,Y 228.618,Z 478.681,A -85,B 0,C 180,E1 21582.699,E2 21582.699} C_VEL
LIN {X 0,Y 226.853,Z 474.649,A -85,B 0,C 180,E1 21585.581,E2 21585.581} C_VEL
LIN {X 0,Y 226.817,Z 474.494,A -85,B 0,C 180,E1 21590.913,E2 21590.913} C_VEL
LIN {X 0,Y 226.831,Z 474.542,A -85,B 0,C 180,E1 21596.209,E2 21596.209} C_VEL
LIN {X 0,Y 226.811,Z 474.489,A -85,B 0,C 180,E1 21601.516,E2 21601.516} C_VEL
LIN {X 0,Y 226.825,Z 474.494,A -85,B 0,C 180,E1 21606.582,E2 21606.582} C_VEL
LIN {X 0,Y 226.814,Z 474.521,A -85,B 0,C 180,E1 21611.958,E2 21611.958} C_VEL
LIN {X 0,Y 226.81,Z 474.479,A -85,B 0,C 180,E1 21616.938,E2 21616.938} C_VEL
LIN {X 0,Y 226.821,Z 474.542,A -85,B 0,C 180,E1 21622.279,E2 21622.279} C_VEL
LIN {X 0,Y 226.797,Z 474.492,A -85,B 0,C 180,E1 21627.575,E2 21627.575} C_VEL
LIN {X 0,Y 226.811,Z 474.5,A -85,B 0,C 180,E1 21632.648,E2 21632.648} C_VEL
LIN {X 0,Y 226.794,Z 474.548,A -85,B 0,C 180,E1 21637.893,E2 21637.893} C_VEL
LIN {X 0,Y 226.858,Z 474.893,A -85,B 0,C 180,E1 21640.615,E2 21640.615} C_VEL
LIN {X 0,Y 228.941,Z 479.689,A -85,B 0,C 180,E1 21643.981,E2 21643.981} C_VEL
LIN {X 0,Y 230.919,Z 484.275,A -85,B 0,C 180,E1 21646.832,E2 21646.832} C_VEL
LIN {X 0,Y 233.646,Z 490.518,A -85,B 0,C 180,E1 21650.384,E2 21650.384} C_VEL
LIN {X 0,Y 237.492,Z 500.839,A -85,B 0,C 180,E1 21655.363,E2 21655.363} C_VEL
LIN {X 0,Y 240.898,Z 511.134,A -85,B 0,C 180,E1 21659.692,E2 21659.692} C_VEL
LIN {X 0,Y 244.281,Z 522.824,A -85,B 0,C 180,E1 21664.026,E2 21664.026} C_VEL
LIN {X 0,Y 247.45,Z 536.099,A -85,B 0,C 180,E1 21668.426,E2 21668.426} C_VEL
LIN {X 0,Y 249.222,Z 545.111,A -85,B 0,C 180,E1 21671.158,E2 21671.158} C_VEL
LIN {X 0,Y 247.732,Z 551.598,A -85,B 0,C 180,E1 21672.501,E2 21672.501} C_VEL
LIN {X 0,Y 254.498,Z 604.172,A -85,B 0,C 180,E1 21675.442,E2 21675.442} C_VEL
LIN {X 0,Y 250.268,Z 691.159,A -85,B 0,C 180,E1 21677.943,E2 21677.943} C_VEL
LIN {X 0,Y 248.857,Z 708.553,A -85,B 0,C 180,E1 21678.887,E2 21678.887} C_VEL
LIN {X 0,Y 246.958,Z 723.871,A -85,B 0,C 180,E1 21680.124,E2 21680.124} C_VEL
LIN {X 0,Y 244.346,Z 739.745,A -85,B 0,C 180,E1 21681.884,E2 21681.884} C_VEL
LIN {X 0,Y 241.507,Z 753.732,A -85,B 0,C 180,E1 21683.939,E2 21683.939} C_VEL
LIN {X 0,Y 238.42,Z 767.121,A -85,B 0,C 180,E1 21686.477,E2 21686.477} C_VEL
LIN {X 0,Y 235.483,Z 778.551,A -85,B 0,C 180,E1 21689.27,E2 21689.27} C_VEL
LIN {X 0,Y 232.725,Z 788.826,A -85,B 0,C 180,E1 21692.462,E2 21692.462} C_VEL
LIN {X 0,Y 230.368,Z 797.487,A -85,B 0,C 180,E1 21695.979,E2 21695.979} C_VEL
LIN {X 0,Y 228.557,Z 804.627,A -85,B 0,C 180,E1 21699.823,E2 21699.823} C_VEL
LIN {X 0,Y 227.451,Z 809.748,A -85,B 0,C 180,E1 21703.732,E2 21703.732} C_VEL
LIN {X 0,Y 227.011,Z 813.334,A -85,B 0,C 180,E1 21707.957,E2 21707.957} C_VEL
LIN {X 0,Y 227.284,Z 814.972,A -85,B 0,C 180,E1 21712.23,E2 21712.23} C_VEL
LIN {X 0,Y 228.251,Z 814.863,A -85,B 0,C 180,E1 21716.259,E2 21716.259} C_VEL
LIN {X 0,Y 230.006,Z 813.013,A -85,B 0,C 180,E1 21720.282,E2 21720.282} C_VEL
LIN {X 0,Y 232.793,Z 809.155,A -85,B 0,C 180,E1 21724.446,E2 21724.446} C_VEL
LIN {X 0,Y 236.202,Z 803.698,A -85,B 0,C 180,E1 21728.172,E2 21728.172} C_VEL
LIN {X 0,Y 240.359,Z 796.355,A -85,B 0,C 180,E1 21731.726,E2 21731.726} C_VEL
LIN {X 0,Y 244.556,Z 788.188,A -85,B 0,C 180,E1 21734.685,E2 21734.685} C_VEL
LIN {X 0,Y 249.289,Z 777.809,A -85,B 0,C 180,E1 21737.56,E2 21737.56} C_VEL
LIN {X 0,Y 254.113,Z 765.889,A -85,B 0,C 180,E1 21740.108,E2 21740.108} C_VEL
LIN {X 0,Y 258.616,Z 752.819,A -85,B 0,C 180,E1 21742.244,E2 21742.244} C_VEL
LIN {X 0,Y 261.725,Z 742.236,A -85,B 0,C 180,E1 21743.622,E2 21743.622} C_VEL
LIN {X 0,Y 262.714,Z 736.598,A -85,B 0,C 180,E1 21744.37,E2 21744.37} C_VEL
LIN {X 0,Y 262.435,Z 722.913,A -85,B 0,C 180,E1 21746.482,E2 21746.482} C_VEL
LIN {X 0,Y 262.552,Z 715.092,A -85,B 0,C 180,E1 21747.394,E2 21747.394} C_VEL
LIN {X 0,Y 262.882,Z 711.98,A -85,B 0,C 180,E1 21747.633,E2 21747.633} C_VEL
LIN {X 0,Y 264.955,Z 695.148,A -85,B 0,C 180,E1 21748.497,E2 21748.497} C_VEL
LIN {X 0,Y 268.933,Z 639.4,A -85,B 0,C 180,E1 21750.08,E2 21750.08} C_VEL
LIN {X 0,Y 270.789,Z 611.266,A -85,B 0,C 180,E1 21750.845,E2 21750.845} C_VEL
LIN {X 0,Y 267.726,Z 585.22,A -85,B 0,C 180,E1 21752.954,E2 21752.954} C_VEL
LIN {X 0,Y 266.033,Z 573.955,A -85,B 0,C 180,E1 21754.032,E2 21754.032} C_VEL
LIN {X 0,Y 260.098,Z 562.694,A -85,B 0,C 180,E1 21756.674,E2 21756.674} C_VEL
LIN {X 0,Y 255.331,Z 554.732,A -85,B 0,C 180,E1 21759.003,E2 21759.003} C_VEL
LIN {X 0,Y 252.708,Z 549.981,A -85,B 0,C 180,E1 21760.588,E2 21760.588} C_VEL
LIN {X 0,Y 250.956,Z 543.188,A -85,B 0,C 180,E1 21764.517,E2 21764.517} C_VEL
LIN {X 0,Y 249.419,Z 537.731,A -85,B 0,C 180,E1 21768.437,E2 21768.437} C_VEL
LIN {X 0,Y 248.179,Z 533.029,A -85,B 0,C 180,E1 21772.592,E2 21772.592} C_VEL
LIN {X 0,Y 247.076,Z 529.574,A -85,B 0,C 180,E1 21776.984,E2 21776.984} C_VEL
LIN {X 0,Y 246.397,Z 526.587,A -85,B 0,C 180,E1 21783.722,E2 21783.722} C_VEL
LIN {X 0,Y 246.54,Z 526.61,A -85,B 0,C 180,E1 21789.335,E2 21789.335} C_VEL
LIN {X 0,Y 247.068,Z 527.618,A -85,B 0,C 180,E1 21792.762,E2 21792.762} C_VEL
LIN {X 0,Y 248.827,Z 531.6,A -85,B 0,C 180,E1 21798.994,E2 21798.994} C_VEL
LIN {X 0,Y 250.475,Z 535.775,A -85,B 0,C 180,E1 21803.029,E2 21803.029} C_VEL
LIN {X 0,Y 252.175,Z 540.192,A -85,B 0,C 180,E1 21806.364,E2 21806.364} C_VEL
LIN {X 0,Y 254.418,Z 546.058,A -85,B 0,C 180,E1 21809.941,E2 21809.941} C_VEL
LIN {X 0,Y 260.057,Z 554.388,A -85,B 0,C 180,E1 21812.827,E2 21812.827} C_VEL
LIN {X 0,Y 265.806,Z 563.283,A -85,B 0,C 180,E1 21815.334,E2 21815.334} C_VEL
LIN {X 0,Y 272.379,Z 574.575,A -85,B 0,C 180,E1 21817.898,E2 21817.898} C_VEL
LIN {X 0,Y 274.018,Z 578.07,A -85,B 0,C 180,E1 21818.522,E2 21818.522} C_VEL
LIN {X 0,Y 274.282,Z 589.015,A -85,B 0,C 180,E1 21819.078,E2 21819.078} C_VEL
LIN {X 0,Y 265.468,Z 722.525,A -85,B 0,C 180,E1 21822.461,E2 21822.461} C_VEL
LIN {X 0,Y 262.973,Z 740.581,A -85,B 0,C 180,E1 21823.213,E2 21823.213} C_VEL
LIN {X 0,Y 259.507,Z 757.422,A -85,B 0,C 180,E1 21824.223,E2 21824.223} C_VEL
LIN {X 0,Y 255.089,Z 774.104,A -85,B 0,C 180,E1 21825.601,E2 21825.601} C_VEL
LIN {X 0,Y 249.907,Z 790.379,A -85,B 0,C 180,E1 21827.406,E2 21827.406} C_VEL
LIN {X 0,Y 244.421,Z 805.282,A -85,B 0,C 180,E1 21829.581,E2 21829.581} C_VEL
LIN {X 0,Y 238.823,Z 819.086,A -85,B 0,C 180,E1 21832.169,E2 21832.169} C_VEL
LIN {X 0,Y 233.216,Z 831.943,A -85,B 0,C 180,E1 21835.236,E2 21835.236} C_VEL
LIN {X 0,Y 227.962,Z 843.737,A -85,B 0,C 180,E1 21838.832,E2 21838.832} C_VEL
LIN {X 0,Y 223.473,Z 854.018,A -85,B 0,C 180,E1 21842.848,E2 21842.848} C_VEL
LIN {X 0,Y 219.981,Z 862.816,A -85,B 0,C 180,E1 21847.319,E2 21847.319} C_VEL
LIN {X 0,Y 217.805,Z 869.903,A -85,B 0,C 180,E1 21852.088,E2 21852.088} C_VEL
LIN {X 0,Y 217.009,Z 875.126,A -85,B 0,C 180,E1 21856.953,E2 21856.953} C_VEL
LIN {X 0,Y 217.383,Z 878.512,A -85,B 0,C 180,E1 21861.803,E2 21861.803} C_VEL
LIN {X 0,Y 218.326,Z 879.964,A -85,B 0,C 180,E1 21866.061,E2 21866.061} C_VEL
LIN {X 0,Y 218.93,Z 879.956,A -85,B 0,C 180,E1 21869.739,E2 21869.739} C_VEL
LIN {X 0,Y 218.682,Z 878.767,A -85,B 0,C 180,E1 21873.146,E2 21873.146} C_VEL
LIN {X 0,Y 217.906,Z 875.928,A -85,B 0,C 180,E1 21877.117,E2 21877.117} C_VEL
LIN {X 0,Y 217.382,Z 871.086,A -85,B 0,C 180,E1 21881.566,E2 21881.566} C_VEL
LIN {X 0,Y 217.631,Z 864.444,A -85,B 0,C 180,E1 21886.002,E2 21886.002} C_VEL
LIN {X 0,Y 218.853,Z 855.98,A -85,B 0,C 180,E1 21890.318,E2 21890.318} C_VEL
LIN {X 0,Y 220.975,Z 846.017,A -85,B 0,C 180,E1 21894.316,E2 21894.316} C_VEL
LIN {X 0,Y 223.842,Z 834.624,A -85,B 0,C 180,E1 21897.971,E2 21897.971} C_VEL
LIN {X 0,Y 227.258,Z 821.77,A -85,B 0,C 180,E1 21901.277,E2 21901.277} C_VEL
LIN {X 0,Y 231.113,Z 807.372,A -85,B 0,C 180,E1 21904.224,E2 21904.224} C_VEL
LIN {X 0,Y 234.979,Z 791.814,A -85,B 0,C 180,E1 21906.716,E2 21906.716} C_VEL
LIN {X 0,Y 238.481,Z 776.195,A -85,B 0,C 180,E1 21908.661,E2 21908.661} C_VEL
LIN {X 0,Y 241.842,Z 758.569,A -85,B 0,C 180,E1 21910.318,E2 21910.318} C_VEL
LIN {X 0,Y 244.509,Z 740.702,A -85,B 0,C 180,E1 21911.521,E2 21911.521} C_VEL
LIN {X 0,Y 246.194,Z 722.54,A -85,B 0,C 180,E1 21912.339,E2 21912.339} C_VEL
LIN {X 0,Y 252.666,Z 581.754,A -85,B 0,C 180,E1 21916.116,E2 21916.116} C_VEL
LIN {X 0,Y 250.95,Z 556.168,A -85,B 0,C 180,E1 21917.287,E2 21917.287} C_VEL
LIN {X 0,Y 245.05,Z 544.155,A -85,B 0,C 180,E1 21918.78,E2 21918.78} C_VEL
LIN {X 0,Y 240.822,Z 529.795,A -85,B 0,C 180,E1 21922.986,E2 21922.986} C_VEL
LIN {X 0,Y 236.599,Z 517.143,A -85,B 0,C 180,E1 21927.254,E2 21927.254} C_VEL
LIN {X 0,Y 232.539,Z 506.326,A -85,B 0,C 180,E1 21931.493,E2 21931.493} C_VEL
LIN {X 0,Y 228.762,Z 496.925,A -85,B 0,C 180,E1 21935.742,E2 21935.742} C_VEL
LIN {X 0,Y 225.034,Z 488.588,A -85,B 0,C 180,E1 21940.265,E2 21940.265} C_VEL
LIN {X 0,Y 222.904,Z 484.171,A -85,B 0,C 180,E1 21943.049,E2 21943.049} C_VEL
LIN {X 0,Y 220.835,Z 479.82,A -85,B 0,C 180,E1 21946.116,E2 21946.116} C_VEL
LIN {X 0,Y 218.901,Z 475.588,A -85,B 0,C 180,E1 21949.739,E2 21949.739} C_VEL
LIN {X 0,Y 218.882,Z 475.506,A -85,B 0,C 180,E1 21954.772,E2 21954.772} C_VEL
LIN {X 0,Y 218.899,Z 475.465,A -85,B 0,C 180,E1 21960.262,E2 21960.262} C_VEL
LIN {X 0,Y 218.876,Z 475.499,A -85,B 0,C 180,E1 21965.768,E2 21965.768} C_VEL
LIN {X 0,Y 218.869,Z 475.487,A -85,B 0,C 180,E1 21971.062,E2 21971.062} C_VEL
LIN {X 0,Y 218.879,Z 475.469,A -85,B 0,C 180,E1 21976.453,E2 21976.453} C_VEL
LIN {X 0,Y 218.87,Z 475.535,A -85,B 0,C 180,E1 21981.972,E2 21981.972} C_VEL
LIN {X 0,Y 218.865,Z 475.475,A -85,B 0,C 180,E1 21987.184,E2 21987.184} C_VEL
LIN {X 0,Y 218.871,Z 475.488,A -85,B 0,C 180,E1 21992.62,E2 21992.62} C_VEL
LIN {X 0,Y 218.9,Z 475.772,A -85,B 0,C 180,E1 21996.494,E2 21996.494} C_VEL
LIN {X 0,Y 221.138,Z 480.688,A -85,B 0,C 180,E1 22000.624,E2 22000.624} C_VEL
LIN {X 0,Y 223.15,Z 485.431,A -85,B 0,C 180,E1 22003.988,E2 22003.988} C_VEL
LIN {X 0,Y 224.837,Z 489.255,A -85,B 0,C 180,E1 22006.459,E2 22006.459} C_VEL
LIN {X 0,Y 227.552,Z 495.83,A -85,B 0,C 180,E1 22010.26,E2 22010.26} C_VEL
LIN {X 0,Y 230.994,Z 505.124,A -85,B 0,C 180,E1 22014.895,E2 22014.895} C_VEL
LIN {X 0,Y 234.301,Z 515.415,A -85,B 0,C 180,E1 22019.339,E2 22019.339} C_VEL
LIN {X 0,Y 237.546,Z 527.042,A -85,B 0,C 180,E1 22023.771,E2 22023.771} C_VEL
LIN {X 0,Y 240.522,Z 539.936,A -85,B 0,C 180,E1 22028.144,E2 22028.144} C_VEL
LIN {X 0,Y 241.934,Z 547.715,A -85,B 0,C 180,E1 22030.567,E2 22030.567} C_VEL
LIN {X 0,Y 241.116,Z 551.553,A -85,B 0,C 180,E1 22031.332,E2 22031.332} C_VEL
LIN {X 0,Y 247.836,Z 605.14,A -85,B 0,C 180,E1 22034.441,E2 22034.441} C_VEL
LIN {X 0,Y 243.447,Z 691.801,A -85,B 0,C 180,E1 22036.982,E2 22036.982} C_VEL
LIN {X 0,Y 241.973,Z 709.21,A -85,B 0,C 180,E1 22037.947,E2 22037.947} C_VEL
LIN {X 0,Y 240.018,Z 724.385,A -85,B 0,C 180,E1 22039.195,E2 22039.195} C_VEL
LIN {X 0,Y 237.412,Z 739.661,A -85,B 0,C 180,E1 22040.913,E2 22040.913} C_VEL
LIN {X 0,Y 234.603,Z 753.2,A -85,B 0,C 180,E1 22042.9,E2 22042.9} C_VEL
LIN {X 0,Y 231.435,Z 766.436,A -85,B 0,C 180,E1 22045.415,E2 22045.415} C_VEL
LIN {X 0,Y 228.356,Z 778.119,A -85,B 0,C 180,E1 22048.243,E2 22048.243} C_VEL
LIN {X 0,Y 225.391,Z 788.641,A -85,B 0,C 180,E1 22051.525,E2 22051.525} C_VEL
LIN {X 0,Y 223.013,Z 797.069,A -85,B 0,C 180,E1 22054.886,E2 22054.886} C_VEL
LIN {X 0,Y 221.083,Z 804.106,A -85,B 0,C 180,E1 22058.583,E2 22058.583} C_VEL
LIN {X 0,Y 219.754,Z 809.753,A -85,B 0,C 180,E1 22062.614,E2 22062.614} C_VEL
LIN {X 0,Y 219.136,Z 813.588,A -85,B 0,C 180,E1 22066.705,E2 22066.705} C_VEL
LIN {X 0,Y 219.221,Z 815.84,A -85,B 0,C 180,E1 22071.119,E2 22071.119} C_VEL
LIN {X 0,Y 220.024,Z 816.289,A -85,B 0,C 180,E1 22075.287,E2 22075.287} C_VEL
LIN {X 0,Y 221.763,Z 814.887,A -85,B 0,C 180,E1 22079.732,E2 22079.732} C_VEL
LIN {X 0,Y 224.34,Z 811.791,A -85,B 0,C 180,E1 22083.856,E2 22083.856} C_VEL
LIN {X 0,Y 227.859,Z 806.7,A -85,B 0,C 180,E1 22087.903,E2 22087.903} C_VEL
LIN {X 0,Y 232.017,Z 800.044,A -85,B 0,C 180,E1 22091.578,E2 22091.578} C_VEL
LIN {X 0,Y 236.603,Z 791.8,A -85,B 0,C 180,E1 22094.888,E2 22094.888} C_VEL
LIN {X 0,Y 241.505,Z 782.018,A -85,B 0,C 180,E1 22097.878,E2 22097.878} C_VEL
LIN {X 0,Y 246.346,Z 771.048,A -85,B 0,C 180,E1 22100.458,E2 22100.458} C_VEL
LIN {X 0,Y 251.458,Z 757.718,A -85,B 0,C 180,E1 22102.866,E2 22102.866} C_VEL
LIN {X 0,Y 255.841,Z 743.978,A -85,B 0,C 180,E1 22104.765,E2 22104.765} C_VEL
LIN {X 0,Y 259.83,Z 728.304,A -85,B 0,C 180,E1 22106.4,E2 22106.4} C_VEL
LIN {X 0,Y 262.77,Z 712.729,A -85,B 0,C 180,E1 22107.587,E2 22107.587} C_VEL
LIN {X 0,Y 262.882,Z 711.98,A -85,B 0,C 180,E1 22107.633,E2 22107.633} C_VEL
LIN {X 0,Y 263.281,Z 704.695,A -85,B 0,C 180,E1 22108.221,E2 22108.221} C_VEL
LIN {X 0,Y 261.459,Z 688.504,A -85,B 0,C 180,E1 22109.825,E2 22109.825} C_VEL
LIN {X 0,Y 261.031,Z 681.087,A -85,B 0,C 180,E1 22110.306,E2 22110.306} C_VEL
LIN {X 0,Y 261.127,Z 678.907,A -85,B 0,C 180,E1 22110.384,E2 22110.384} C_VEL
LIN {X 0,Y 265.914,Z 612.846,A -85,B 0,C 180,E1 22112.175,E2 22112.175} C_VEL
LIN {X 0,Y 263.112,Z 587.146,A -85,B 0,C 180,E1 22114.328,E2 22114.328} C_VEL
LIN {X 0,Y 261.904,Z 578.765,A -85,B 0,C 180,E1 22115.168,E2 22115.168} C_VEL
LIN {X 0,Y 256.825,Z 568.809,A -85,B 0,C 180,E1 22117.571,E2 22117.571} C_VEL
LIN {X 0,Y 252.417,Z 561.206,A -85,B 0,C 180,E1 22119.841,E2 22119.841} C_VEL
LIN {X 0,Y 248.471,Z 554.729,A -85,B 0,C 180,E1 22122.131,E2 22122.131} C_VEL
LIN {X 0,Y 245.507,Z 549.453,A -85,B 0,C 180,E1 22124.286,E2 22124.286} C_VEL
LIN {X 0,Y 243.977,Z 543.723,A -85,B 0,C 180,E1 22128.415,E2 22128.415} C_VEL
LIN {X 0,Y 242.767,Z 538.892,A -85,B 0,C 180,E1 22132.783,E2 22132.783} C_VEL
LIN {X 0,Y 241.785,Z 535.546,A -85,B 0,C 180,E1 22137.155,E2 22137.155} C_VEL
LIN {X 0,Y 241.25,Z 532.706,A -85,B 0,C 180,E1 22143.802,E2 22143.802} C_VEL
LIN {X 0,Y 241.462,Z 532.795,A -85,B 0,C 180,E1 22149.534,E2 22149.534} C_VEL
LIN {X 0,Y 241.942,Z 533.794,A -85,B 0,C 180,E1 22152.762,E2 22152.762} C_VEL
LIN {X 0,Y 243.562,Z 537.468,A -85,B 0,C 180,E1 22158.675,E2 22158.675} C_VEL
LIN {X 0,Y 245.159,Z 541.699,A -85,B 0,C 180,E1 22162.822,E2 22162.822} C_VEL
LIN {X 0,Y 246.81,Z 546.113,A -85,B 0,C 180,E1 22166.204,E2 22166.204} C_VEL
LIN {X 0,Y 251.736,Z 553.07,A -85,B 0,C 180,E1 22169.309,E2 22169.309} C_VEL
LIN {X 0,Y 257.416,Z 561.47,A -85,B 0,C 180,E1 22172.215,E2 22172.215} C_VEL
LIN {X 0,Y 263.213,Z 570.685,A -85,B 0,C 180,E1 22174.835,E2 22174.835} C_VEL
LIN {X 0,Y 269.328,Z 581.869,A -85,B 0,C 180,E1 22177.338,E2 22177.338} C_VEL
LIN {X 0,Y 269.427,Z 590.151,A -85,B 0,C 180,E1 22177.75,E2 22177.75} C_VEL
LIN {X 0,Y 260.347,Z 721.9,A -85,B 0,C 180,E1 22181.11,E2 22181.11} C_VEL
LIN {X 0,Y 257.766,Z 739.915,A -85,B 0,C 180,E1 22181.862,E2 22181.862} C_VEL
LIN {X 0,Y 253.984,Z 757.492,A -85,B 0,C 180,E1 22182.927,E2 22182.927} C_VEL
LIN {X 0,Y 249.41,Z 773.933,A -85,B 0,C 180,E1 22184.309,E2 22184.309} C_VEL
LIN {X 0,Y 244.214,Z 789.474,A -85,B 0,C 180,E1 22186.056,E2 22186.056} C_VEL
LIN {X 0,Y 238.309,Z 804.751,A -85,B 0,C 180,E1 22188.316,E2 22188.316} C_VEL
LIN {X 0,Y 232.213,Z 819.001,A -85,B 0,C 180,E1 22191.05,E2 22191.05} C_VEL
LIN {X 0,Y 226.148,Z 832.137,A -85,B 0,C 180,E1 22194.296,E2 22194.296} C_VEL
LIN {X 0,Y 220.65,Z 843.706,A -85,B 0,C 180,E1 22197.983,E2 22197.983} C_VEL
LIN {X 0,Y 215.811,Z 853.976,A -85,B 0,C 180,E1 22202.239,E2 22202.239} C_VEL
LIN {X 0,Y 212.093,Z 862.687,A -85,B 0,C 180,E1 22206.966,E2 22206.966} C_VEL
LIN {X 0,Y 209.827,Z 869.578,A -85,B 0,C 180,E1 22211.957,E2 22211.957} C_VEL
LIN {X 0,Y 209.031,Z 874.548,A -85,B 0,C 180,E1 22217.008,E2 22217.008} C_VEL
LIN {X 0,Y 209.469,Z 877.651,A -85,B 0,C 180,E1 22222.044,E2 22222.044} C_VEL
LIN {X 0,Y 210.483,Z 878.889,A -85,B 0,C 180,E1 22226.46,E2 22226.46} C_VEL
LIN {X 0,Y 211.044,Z 878.668,A -85,B 0,C 180,E1 22230,E2 22230} C_VEL
LIN {X 0,Y 210.687,Z 877.324,A -85,B 0,C 180,E1 22233.538,E2 22233.538} C_VEL
LIN {X 0,Y 209.819,Z 874.058,A -85,B 0,C 180,E1 22237.944,E2 22237.944} C_VEL
LIN {X 0,Y 209.404,Z 869.08,A -85,B 0,C 180,E1 22242.408,E2 22242.408} C_VEL
LIN {X 0,Y 209.821,Z 862.307,A -85,B 0,C 180,E1 22246.899,E2 22246.899} C_VEL
LIN {X 0,Y 211.27,Z 853.561,A -85,B 0,C 180,E1 22251.372,E2 22251.372} C_VEL
LIN {X 0,Y 213.665,Z 843.308,A -85,B 0,C 180,E1 22255.501,E2 22255.501} C_VEL
LIN {X 0,Y 216.813,Z 831.577,A -85,B 0,C 180,E1 22259.264,E2 22259.264} C_VEL
LIN {X 0,Y 220.554,Z 818.29,A -85,B 0,C 180,E1 22262.648,E2 22262.648} C_VEL
LIN {X 0,Y 224.503,Z 803.912,A -85,B 0,C 180,E1 22265.536,E2 22265.536} C_VEL
LIN {X 0,Y 228.415,Z 788.591,A -85,B 0,C 180,E1 22267.954,E2 22267.954} C_VEL
LIN {X 0,Y 232.106,Z 772.356,A -85,B 0,C 180,E1 22269.935,E2 22269.935} C_VEL
LIN {X 0,Y 235.403,Z 755.237,A -85,B 0,C 180,E1 22271.499,E2 22271.499} C_VEL
LIN {X 0,Y 237.987,Z 737.285,A -85,B 0,C 180,E1 22272.657,E2 22272.657} C_VEL
LIN {X 0,Y 239.552,Z 719.101,A -85,B 0,C 180,E1 22273.427,E2 22273.427} C_VEL
LIN {X 0,Y 246.07,Z 582.39,A -85,B 0,C 180,E1 22277.159,E2 22277.159} C_VEL
LIN {X 0,Y 244.505,Z 559.044,A -85,B 0,C 180,E1 22278.277,E2 22278.277} C_VEL
LIN {X 0,Y 237.314,Z 544.541,A -85,B 0,C 180,E1 22280.178,E2 22280.178} C_VEL
LIN {X 0,Y 233.282,Z 531.031,A -85,B 0,C 180,E1 22284.346,E2 22284.346} C_VEL
LIN {X 0,Y 229.156,Z 518.703,A -85,B 0,C 180,E1 22288.782,E2 22288.782} C_VEL
LIN {X 0,Y 225.231,Z 508.248,A -85,B 0,C 180,E1 22293.164,E2 22293.164} C_VEL
LIN {X 0,Y 221.808,Z 500.09,A -85,B 0,C 180,E1 22297.191,E2 22297.191} C_VEL
LIN {X 0,Y 219.274,Z 494.049,A -85,B 0,C 180,E1 22300.557,E2 22300.557} C_VEL
LIN {X 0,Y 216.961,Z 489.307,A -85,B 0,C 180,E1 22303.674,E2 22303.674} C_VEL
LIN {X 0,Y 215.146,Z 485.351,A -85,B 0,C 180,E1 22306.564,E2 22306.564} C_VEL
LIN {X 0,Y 213.025,Z 480.979,A -85,B 0,C 180,E1 22310.273,E2 22310.273} C_VEL
LIN {X 0,Y 210.952,Z 476.599,A -85,B 0,C 180,E1 22315.106,E2 22315.106} C_VEL
LIN {X 0,Y 210.946,Z 476.455,A -85,B 0,C 180,E1 22320.544,E2 22320.544} C_VEL
LIN {X 0,Y 210.943,Z 476.479,A -85,B 0,C 180,E1 22325.986,E2 22325.986} C_VEL
LIN {X 0,Y 210.928,Z 476.477,A -85,B 0,C 180,E1 22331.207,E2 22331.207} C_VEL
LIN {X 0,Y 210.939,Z 476.456,A -85,B 0,C 180,E1 22336.524,E2 22336.524} C_VEL
LIN {X 0,Y 210.932,Z 476.524,A -85,B 0,C 180,E1 22341.993,E2 22341.993} C_VEL
LIN {X 0,Y 210.922,Z 476.464,A -85,B 0,C 180,E1 22347.376,E2 22347.376} C_VEL
LIN {X 0,Y 210.981,Z 476.875,A -85,B 0,C 180,E1 22351.326,E2 22351.326} C_VEL
LIN {X 0,Y 213.35,Z 481.952,A -85,B 0,C 180,E1 22356.736,E2 22356.736} C_VEL
LIN {X 0,Y 215.403,Z 486.397,A -85,B 0,C 180,E1 22360.531,E2 22360.531} C_VEL
LIN {X 0,Y 217.26,Z 490.766,A -85,B 0,C 180,E1 22363.735,E2 22363.735} C_VEL
LIN {X 0,Y 219.036,Z 495.046,A -85,B 0,C 180,E1 22366.537,E2 22366.537} C_VEL
LIN {X 0,Y 221.478,Z 501.135,A -85,B 0,C 180,E1 22370.129,E2 22370.129} C_VEL
LIN {X 0,Y 224.664,Z 509.961,A -85,B 0,C 180,E1 22374.65,E2 22374.65} C_VEL
LIN {X 0,Y 227.795,Z 520.018,A -85,B 0,C 180,E1 22379.099,E2 22379.099} C_VEL
LIN {X 0,Y 230.826,Z 531.279,A -85,B 0,C 180,E1 22383.502,E2 22383.502} C_VEL
LIN {X 0,Y 233.613,Z 543.853,A -85,B 0,C 180,E1 22387.874,E2 22387.874} C_VEL
LIN {X 0,Y 234.681,Z 550.378,A -85,B 0,C 180,E1 22389.942,E2 22389.942} C_VEL
LIN {X 0,Y 234.789,Z 553.169,A -85,B 0,C 180,E1 22390.216,E2 22390.216} C_VEL
LIN {X 0,Y 241.22,Z 606.186,A -85,B 0,C 180,E1 22393.396,E2 22393.396} C_VEL
LIN {X 0,Y 236.676,Z 692.331,A -85,B 0,C 180,E1 22395.972,E2 22395.972} C_VEL
LIN {X 0,Y 235.134,Z 709.784,A -85,B 0,C 180,E1 22396.959,E2 22396.959} C_VEL
LIN {X 0,Y 233.084,Z 725.079,A -85,B 0,C 180,E1 22398.243,E2 22398.243} C_VEL
LIN {X 0,Y 230.365,Z 740.378,A -85,B 0,C 180,E1 22400.002,E2 22400.002} C_VEL
LIN {X 0,Y 227.433,Z 753.951,A -85,B 0,C 180,E1 22402.039,E2 22402.039} C_VEL
LIN {X 0,Y 224.122,Z 767.218,A -85,B 0,C 180,E1 22404.624,E2 22404.624} C_VEL
LIN {X 0,Y 221.03,Z 778.489,A -85,B 0,C 180,E1 22407.407,E2 22407.407} C_VEL
LIN {X 0,Y 217.897,Z 789.14,A -85,B 0,C 180,E1 22410.788,E2 22410.788} C_VEL
LIN {X 0,Y 215.205,Z 798.266,A -85,B 0,C 180,E1 22414.53,E2 22414.53} C_VEL
LIN {X 0,Y 213.083,Z 805.718,A -85,B 0,C 180,E1 22418.635,E2 22418.635} C_VEL
LIN {X 0,Y 211.765,Z 811.248,A -85,B 0,C 180,E1 22422.821,E2 22422.821} C_VEL
LIN {X 0,Y 211.172,Z 815.133,A -85,B 0,C 180,E1 22427.355,E2 22427.355} C_VEL
LIN {X 0,Y 211.398,Z 817.194,A -85,B 0,C 180,E1 22431.94,E2 22431.94} C_VEL
LIN {X 0,Y 212.506,Z 817.342,A -85,B 0,C 180,E1 22436.623,E2 22436.623} C_VEL
LIN {X 0,Y 214.571,Z 815.655,A -85,B 0,C 180,E1 22441.147,E2 22441.147} C_VEL
LIN {X 0,Y 217.522,Z 812.163,A -85,B 0,C 180,E1 22445.392,E2 22445.392} C_VEL
LIN {X 0,Y 221.472,Z 806.766,A -85,B 0,C 180,E1 22449.535,E2 22449.535} C_VEL
LIN {X 0,Y 226.041,Z 799.655,A -85,B 0,C 180,E1 22453.284,E2 22453.284} C_VEL
LIN {X 0,Y 231.047,Z 791.077,A -85,B 0,C 180,E1 22456.637,E2 22456.637} C_VEL
LIN {X 0,Y 236.324,Z 780.801,A -85,B 0,C 180,E1 22459.659,E2 22459.659} C_VEL
LIN {X 0,Y 241.761,Z 768.766,A -85,B 0,C 180,E1 22462.363,E2 22462.363} C_VEL
LIN {X 0,Y 246.766,Z 755.762,A -85,B 0,C 180,E1 22464.59,E2 22464.59} C_VEL
LIN {X 0,Y 251.431,Z 741.119,A -85,B 0,C 180,E1 22466.509,E2 22466.509} C_VEL
LIN {X 0,Y 255.113,Z 726.436,A -85,B 0,C 180,E1 22467.955,E2 22467.955} C_VEL
LIN {X 0,Y 258.181,Z 709.763,A -85,B 0,C 180,E1 22469.151,E2 22469.151} C_VEL
LIN {X 0,Y 260.084,Z 693.47,A -85,B 0,C 180,E1 22469.93,E2 22469.93} C_VEL
LIN {X 0,Y 261.127,Z 678.907,A -85,B 0,C 180,E1 22470.384,E2 22470.384} C_VEL
LIN {X 0,Y 261.079,Z 671.338,A -85,B 0,C 180,E1 22470.768,E2 22470.768} C_VEL
LIN {X 0,Y 258.868,Z 651.569,A -85,B 0,C 180,E1 22472.415,E2 22472.415} C_VEL
LIN {X 0,Y 258.946,Z 645.059,A -85,B 0,C 180,E1 22472.721,E2 22472.721} C_VEL
LIN {X 0,Y 261.199,Z 614.372,A -85,B 0,C 180,E1 22473.561,E2 22473.561} C_VEL
LIN {X 0,Y 258.615,Z 588.338,A -85,B 0,C 180,E1 22475.82,E2 22475.82} C_VEL
LIN {X 0,Y 257.895,Z 583.53,A -85,B 0,C 180,E1 22476.342,E2 22476.342} C_VEL
LIN {X 0,Y 253.017,Z 573.879,A -85,B 0,C 180,E1 22478.802,E2 22478.802} C_VEL
LIN {X 0,Y 249.411,Z 567.378,A -85,B 0,C 180,E1 22480.808,E2 22480.808} C_VEL
LIN {X 0,Y 245.971,Z 561.534,A -85,B 0,C 180,E1 22482.92,E2 22482.92} C_VEL
LIN {X 0,Y 242.333,Z 555.641,A -85,B 0,C 180,E1 22485.422,E2 22485.422} C_VEL
LIN {X 0,Y 238.592,Z 549.565,A -85,B 0,C 180,E1 22488.64,E2 22488.64} C_VEL
LIN {X 0,Y 237.459,Z 545.53,A -85,B 0,C 180,E1 22492.256,E2 22492.256} C_VEL
LIN {X 0,Y 236.582,Z 541.643,A -85,B 0,C 180,E1 22497.092,E2 22497.092} C_VEL
LIN {X 0,Y 236.1,Z 538.822,A -85,B 0,C 180,E1 22503.885,E2 22503.885} C_VEL
LIN {X 0,Y 236.386,Z 538.986,A -85,B 0,C 180,E1 22509.759,E2 22509.759} C_VEL
LIN {X 0,Y 236.815,Z 539.974,A -85,B 0,C 180,E1 22512.761,E2 22512.761} C_VEL
LIN {X 0,Y 238.353,Z 543.589,A -85,B 0,C 180,E1 22518.591,E2 22518.591} C_VEL
LIN {X 0,Y 239.933,Z 547.258,A -85,B 0,C 180,E1 22522.156,E2 22522.156} C_VEL
LIN {X 0,Y 245.899,Z 555.342,A -85,B 0,C 180,E1 22526.569,E2 22526.569} C_VEL
LIN {X 0,Y 251,Z 562.703,A -85,B 0,C 180,E1 22529.6,E2 22529.6} C_VEL
LIN {X 0,Y 255.64,Z 569.869,A -85,B 0,C 180,E1 22532.003,E2 22532.003} C_VEL
LIN {X 0,Y 261.74,Z 580.289,A -85,B 0,C 180,E1 22534.826,E2 22534.826} C_VEL
LIN {X 0,Y 264.782,Z 586.351,A -85,B 0,C 180,E1 22536.15,E2 22536.15} C_VEL
LIN {X 0,Y 264.662,Z 592.139,A -85,B 0,C 180,E1 22536.396,E2 22536.396} C_VEL
LIN {X 0,Y 255.377,Z 721.277,A -85,B 0,C 180,E1 22539.706,E2 22539.706} C_VEL
LIN {X 0,Y 252.682,Z 739.382,A -85,B 0,C 180,E1 22540.463,E2 22540.463} C_VEL
LIN {X 0,Y 248.92,Z 756.313,A -85,B 0,C 180,E1 22541.485,E2 22541.485} C_VEL
LIN {X 0,Y 244.173,Z 772.83,A -85,B 0,C 180,E1 22542.863,E2 22542.863} C_VEL
LIN {X 0,Y 238.766,Z 788.421,A -85,B 0,C 180,E1 22544.611,E2 22544.611} C_VEL
LIN {X 0,Y 232.59,Z 803.705,A -85,B 0,C 180,E1 22546.882,E2 22546.882} C_VEL
LIN {X 0,Y 226.182,Z 817.91,A -85,B 0,C 180,E1 22549.638,E2 22549.638} C_VEL
LIN {X 0,Y 219.995,Z 830.589,A -85,B 0,C 180,E1 22552.809,E2 22552.809} C_VEL
LIN {X 0,Y 214.089,Z 842.241,A -85,B 0,C 180,E1 22556.558,E2 22556.558} C_VEL
LIN {X 0,Y 208.978,Z 852.322,A -85,B 0,C 180,E1 22560.79,E2 22560.79} C_VEL
LIN {X 0,Y 204.924,Z 860.889,A -85,B 0,C 180,E1 22565.498,E2 22565.498} C_VEL
LIN {X 0,Y 202.238,Z 867.903,A -85,B 0,C 180,E1 22570.656,E2 22570.656} C_VEL
LIN {X 0,Y 201.109,Z 872.994,A -85,B 0,C 180,E1 22575.901,E2 22575.901} C_VEL
LIN {X 0,Y 201.365,Z 876.276,A -85,B 0,C 180,E1 22581.156,E2 22581.156} C_VEL
LIN {X 0,Y 202.449,Z 877.671,A -85,B 0,C 180,E1 22586.057,E2 22586.057} C_VEL
LIN {X 0,Y 203.118,Z 877.49,A -85,B 0,C 180,E1 22589.718,E2 22589.718} C_VEL
LIN {X 0,Y 202.844,Z 876.328,A -85,B 0,C 180,E1 22593.109,E2 22593.109} C_VEL
LIN {X 0,Y 201.968,Z 873.396,A -85,B 0,C 180,E1 22597.396,E2 22597.396} C_VEL
LIN {X 0,Y 201.455,Z 868.548,A -85,B 0,C 180,E1 22602.112,E2 22602.112} C_VEL
LIN {X 0,Y 201.854,Z 861.634,A -85,B 0,C 180,E1 22606.993,E2 22606.993} C_VEL
LIN {X 0,Y 203.366,Z 852.894,A -85,B 0,C 180,E1 22611.686,E2 22611.686} C_VEL
LIN {X 0,Y 206.029,Z 842.096,A -85,B 0,C 180,E1 22616.208,E2 22616.208} C_VEL
LIN {X 0,Y 209.357,Z 830.308,A -85,B 0,C 180,E1 22620.098,E2 22620.098} C_VEL
LIN {X 0,Y 213.136,Z 817.494,A -85,B 0,C 180,E1 22623.451,E2 22623.451} C_VEL
LIN {X 0,Y 217.248,Z 803.113,A -85,B 0,C 180,E1 22626.421,E2 22626.421} C_VEL
LIN {X 0,Y 221.314,Z 787.796,A -85,B 0,C 180,E1 22628.902,E2 22628.902} C_VEL
LIN {X 0,Y 225.139,Z 771.597,A -85,B 0,C 180,E1 22630.925,E2 22630.925} C_VEL
LIN {X 0,Y 228.556,Z 754.456,A -85,B 0,C 180,E1 22632.524,E2 22632.524} C_VEL
LIN {X 0,Y 231.203,Z 736.609,A -85,B 0,C 180,E1 22633.698,E2 22633.698} C_VEL
LIN {X 0,Y 232.83,Z 718.278,A -85,B 0,C 180,E1 22634.489,E2 22634.489} C_VEL
LIN {X 0,Y 239.577,Z 583.27,A -85,B 0,C 180,E1 22638.247,E2 22638.247} C_VEL
LIN {X 0,Y 238.218,Z 562.055,A -85,B 0,C 180,E1 22639.297,E2 22639.297} C_VEL
LIN {X 0,Y 229.434,Z 544.52,A -85,B 0,C 180,E1 22641.77,E2 22641.77} C_VEL
LIN {X 0,Y 225.656,Z 531.899,A -85,B 0,C 180,E1 22645.954,E2 22645.954} C_VEL
LIN {X 0,Y 221.879,Z 520.639,A -85,B 0,C 180,E1 22650.285,E2 22650.285} C_VEL
LIN {X 0,Y 218.166,Z 510.595,A -85,B 0,C 180,E1 22654.773,E2 22654.773} C_VEL
LIN {X 0,Y 214.615,Z 502.237,A -85,B 0,C 180,E1 22659.264,E2 22659.264} C_VEL
LIN {X 0,Y 212.844,Z 498.352,A -85,B 0,C 180,E1 22661.655,E2 22661.655} C_VEL
LIN {X 0,Y 211.257,Z 494.762,A -85,B 0,C 180,E1 22664.068,E2 22664.068} C_VEL
LIN {X 0,Y 209.656,Z 491.128,A -85,B 0,C 180,E1 22666.767,E2 22666.767} C_VEL
LIN {X 0,Y 207.567,Z 486.772,A -85,B 0,C 180,E1 22670.574,E2 22670.574} C_VEL
LIN {X 0,Y 205.199,Z 482.1,A -85,B 0,C 180,E1 22675.809,E2 22675.809} C_VEL
LIN {X 0,Y 203.018,Z 477.634,A -85,B 0,C 180,E1 22683.671,E2 22683.671} C_VEL
LIN {X 0,Y 202.99,Z 477.439,A -85,B 0,C 180,E1 22689.069,E2 22689.069} C_VEL
LIN {X 0,Y 203.017,Z 477.472,A -85,B 0,C 180,E1 22694.548,E2 22694.548} C_VEL
LIN {X 0,Y 203.005,Z 477.496,A -85,B 0,C 180,E1 22700.469,E2 22700.469} C_VEL
LIN {X 0,Y 203.079,Z 478.063,A -85,B 0,C 180,E1 22703.504,E2 22703.504} C_VEL
LIN {X 0,Y 205.513,Z 482.878,A -85,B 0,C 180,E1 22711.372,E2 22711.372} C_VEL
LIN {X 0,Y 207.706,Z 487.583,A -85,B 0,C 180,E1 22716.494,E2 22716.494} C_VEL
LIN {X 0,Y 209.692,Z 492.1,A -85,B 0,C 180,E1 22720.428,E2 22720.428} C_VEL
LIN {X 0,Y 211.31,Z 495.892,A -85,B 0,C 180,E1 22723.323,E2 22723.323} C_VEL
LIN {X 0,Y 213.252,Z 500.798,A -85,B 0,C 180,E1 22726.614,E2 22726.614} C_VEL
LIN {X 0,Y 216.238,Z 508.517,A -85,B 0,C 180,E1 22731.16,E2 22731.16} C_VEL
LIN {X 0,Y 219.436,Z 518.263,A -85,B 0,C 180,E1 22736.026,E2 22736.026} C_VEL
LIN {X 0,Y 222.503,Z 529.016,A -85,B 0,C 180,E1 22740.671,E2 22740.671} C_VEL
LIN {X 0,Y 225.156,Z 540.223,A -85,B 0,C 180,E1 22744.948,E2 22744.948} C_VEL
LIN {X 0,Y 227.426,Z 551.162,A -85,B 0,C 180,E1 22748.617,E2 22748.617} C_VEL
LIN {X 0,Y 228.51,Z 554.326,A -85,B 0,C 180,E1 22748.998,E2 22748.998} C_VEL
LIN {X 0,Y 234.69,Z 607.23,A -85,B 0,C 180,E1 22752.293,E2 22752.293} C_VEL
LIN {X 0,Y 229.982,Z 692.861,A -85,B 0,C 180,E1 22754.903,E2 22754.903} C_VEL
LIN {X 0,Y 228.382,Z 710.252,A -85,B 0,C 180,E1 22755.905,E2 22755.905} C_VEL
LIN {X 0,Y 226.217,Z 725.773,A -85,B 0,C 180,E1 22757.232,E2 22757.232} C_VEL
LIN {X 0,Y 223.323,Z 741.374,A -85,B 0,C 180,E1 22759.071,E2 22759.071} C_VEL
LIN {X 0,Y 220.142,Z 755.387,A -85,B 0,C 180,E1 22761.248,E2 22761.248} C_VEL
LIN {X 0,Y 216.698,Z 768.57,A -85,B 0,C 180,E1 22763.908,E2 22763.908} C_VEL
LIN {X 0,Y 213.477,Z 779.768,A -85,B 0,C 180,E1 22766.778,E2 22766.778} C_VEL
LIN {X 0,Y 210.212,Z 790.369,A -85,B 0,C 180,E1 22770.272,E2 22770.272} C_VEL
LIN {X 0,Y 207.407,Z 799.46,A -85,B 0,C 180,E1 22774.146,E2 22774.146} C_VEL
LIN {X 0,Y 205.19,Z 806.932,A -85,B 0,C 180,E1 22778.429,E2 22778.429} C_VEL
LIN {X 0,Y 203.835,Z 812.417,A -85,B 0,C 180,E1 22782.752,E2 22782.752} C_VEL
LIN {X 0,Y 203.239,Z 816.305,A -85,B 0,C 180,E1 22787.463,E2 22787.463} C_VEL
LIN {X 0,Y 203.514,Z 818.376,A -85,B 0,C 180,E1 22792.228,E2 22792.228} C_VEL
LIN {X 0,Y 204.703,Z 818.55,A -85,B 0,C 180,E1 22797.016,E2 22797.016} C_VEL
LIN {X 0,Y 206.944,Z 816.895,A -85,B 0,C 180,E1 22801.749,E2 22801.749} C_VEL
LIN {X 0,Y 210.116,Z 813.421,A -85,B 0,C 180,E1 22806.161,E2 22806.161} C_VEL
LIN {X 0,Y 214.314,Z 808.084,A -85,B 0,C 180,E1 22810.427,E2 22810.427} C_VEL
LIN {X 0,Y 219.146,Z 801.059,A -85,B 0,C 180,E1 22814.272,E2 22814.272} C_VEL
LIN {X 0,Y 224.456,Z 792.47,A -85,B 0,C 180,E1 22817.728,E2 22817.728} C_VEL
LIN {X 0,Y 229.866,Z 782.563,A -85,B 0,C 180,E1 22820.737,E2 22820.737} C_VEL
LIN {X 0,Y 235.362,Z 771.063,A -85,B 0,C 180,E1 22823.408,E2 22823.408} C_VEL
LIN {X 0,Y 240.474,Z 758.739,A -85,B 0,C 180,E1 22825.622,E2 22825.622} C_VEL
LIN {X 0,Y 245.266,Z 744.725,A -85,B 0,C 180,E1 22827.55,E2 22827.55} C_VEL
LIN {X 0,Y 249.414,Z 729.633,A -85,B 0,C 180,E1 22829.127,E2 22829.127} C_VEL
LIN {X 0,Y 252.614,Z 713.927,A -85,B 0,C 180,E1 22830.328,E2 22830.328} C_VEL
LIN {X 0,Y 254.914,Z 696.976,A -85,B 0,C 180,E1 22831.216,E2 22831.216} C_VEL
LIN {X 0,Y 258.321,Z 653.072,A -85,B 0,C 180,E1 22832.507,E2 22832.507} C_VEL
LIN {X 0,Y 258.946,Z 645.059,A -85,B 0,C 180,E1 22832.721,E2 22832.721} C_VEL
LIN {X 0,Y 259.054,Z 636.381,A -85,B 0,C 180,E1 22833.133,E2 22833.133} C_VEL
LIN {X 0,Y 257.812,Z 623.887,A -85,B 0,C 180,E1 22834.193,E2 22834.193} C_VEL
LIN {X 0,Y 256.34,Z 611.493,A -85,B 0,C 180,E1 22835.367,E2 22835.367} C_VEL
LIN {X 0,Y 254.101,Z 588.491,A -85,B 0,C 180,E1 22837.5,E2 22837.5} C_VEL
LIN {X 0,Y 249.733,Z 579.622,A -85,B 0,C 180,E1 22839.859,E2 22839.859} C_VEL
LIN {X 0,Y 245.121,Z 570.904,A -85,B 0,C 180,E1 22842.676,E2 22842.676} C_VEL
LIN {X 0,Y 240.272,Z 562.838,A -85,B 0,C 180,E1 22846.094,E2 22846.094} C_VEL
LIN {X 0,Y 236.229,Z 556.316,A -85,B 0,C 180,E1 22849.636,E2 22849.636} C_VEL
LIN {X 0,Y 232.143,Z 550.148,A -85,B 0,C 180,E1 22854.438,E2 22854.438} C_VEL
LIN {X 0,Y 231.379,Z 547.741,A -85,B 0,C 180,E1 22857.027,E2 22857.027} C_VEL
LIN {X 0,Y 230.96,Z 544.947,A -85,B 0,C 180,E1 22863.971,E2 22863.971} C_VEL
LIN {X 0,Y 231.316,Z 545.181,A -85,B 0,C 180,E1 22869.956,E2 22869.956} C_VEL
LIN {X 0,Y 231.704,Z 546.273,A -85,B 0,C 180,E1 22872.967,E2 22872.967} C_VEL
LIN {X 0,Y 232.713,Z 548.35,A -85,B 0,C 180,E1 22875.96,E2 22875.96} C_VEL
LIN {X 0,Y 234.904,Z 550.996,A -85,B 0,C 180,E1 22878.616,E2 22878.616} C_VEL
LIN {X 0,Y 238.407,Z 555.259,A -85,B 0,C 180,E1 22881.916,E2 22881.916} C_VEL
LIN {X 0,Y 243.777,Z 562.65,A -85,B 0,C 180,E1 22885.966,E2 22885.966} C_VEL
LIN {X 0,Y 248.461,Z 569.605,A -85,B 0,C 180,E1 22888.875,E2 22888.875} C_VEL
LIN {X 0,Y 253.77,Z 578.052,A -85,B 0,C 180,E1 22891.735,E2 22891.735} C_VEL
LIN {X 0,Y 259.866,Z 589.262,A -85,B 0,C 180,E1 22894.644,E2 22894.644} C_VEL
LIN {X 0,Y 260.375,Z 590.738,A -85,B 0,C 180,E1 22894.898,E2 22894.898} C_VEL
LIN {X 0,Y 250.565,Z 720.655,A -85,B 0,C 180,E1 22898.246,E2 22898.246} C_VEL
LIN {X 0,Y 247.784,Z 738.705,A -85,B 0,C 180,E1 22899.001,E2 22899.001} C_VEL
LIN {X 0,Y 244.024,Z 755.136,A -85,B 0,C 180,E1 22899.986,E2 22899.986} C_VEL
LIN {X 0,Y 239.116,Z 771.674,A -85,B 0,C 180,E1 22901.351,E2 22901.351} C_VEL
LIN {X 0,Y 233.479,Z 787.366,A -85,B 0,C 180,E1 22903.101,E2 22903.101} C_VEL
LIN {X 0,Y 227.316,Z 802.051,A -85,B 0,C 180,E1 22905.271,E2 22905.271} C_VEL
LIN {X 0,Y 220.622,Z 816.233,A -85,B 0,C 180,E1 22908.008,E2 22908.008} C_VEL
LIN {X 0,Y 213.798,Z 829.501,A -85,B 0,C 180,E1 22911.352,E2 22911.352} C_VEL
LIN {X 0,Y 207.677,Z 840.785,A -85,B 0,C 180,E1 22915.046,E2 22915.046} C_VEL
LIN {X 0,Y 202.127,Z 850.97,A -85,B 0,C 180,E1 22919.397,E2 22919.397} C_VEL
LIN {X 0,Y 197.682,Z 859.529,A -85,B 0,C 180,E1 22924.216,E2 22924.216} C_VEL
LIN {X 0,Y 194.62,Z 866.578,A -85,B 0,C 180,E1 22929.553,E2 22929.553} C_VEL
LIN {X 0,Y 193.211,Z 871.699,A -85,B 0,C 180,E1 22935.005,E2 22935.005} C_VEL
LIN {X 0,Y 193.313,Z 875.004,A -85,B 0,C 180,E1 22940.474,E2 22940.474} C_VEL
LIN {X 0,Y 194.383,Z 876.441,A -85,B 0,C 180,E1 22945.575,E2 22945.575} C_VEL
LIN {X 0,Y 195.184,Z 876.309,A -85,B 0,C 180,E1 22949.414,E2 22949.414} C_VEL
LIN {X 0,Y 194.949,Z 875.171,A -85,B 0,C 180,E1 22952.94,E2 22952.94} C_VEL
LIN {X 0,Y 194.023,Z 872.244,A -85,B 0,C 180,E1 22957.403,E2 22957.403} C_VEL
LIN {X 0,Y 193.492,Z 867.289,A -85,B 0,C 180,E1 22962.409,E2 22962.409} C_VEL
LIN {X 0,Y 193.984,Z 860.235,A -85,B 0,C 180,E1 22967.533,E2 22967.533} C_VEL
LIN {X 0,Y 195.592,Z 851.648,A -85,B 0,C 180,E1 22972.293,E2 22972.293} C_VEL
LIN {X 0,Y 198.327,Z 841.178,A -85,B 0,C 180,E1 22976.832,E2 22976.832} C_VEL
LIN {X 0,Y 201.668,Z 829.889,A -85,B 0,C 180,E1 22980.709,E2 22980.709} C_VEL
LIN {X 0,Y 205.761,Z 816.66,A -85,B 0,C 180,E1 22984.311,E2 22984.311} C_VEL
LIN {X 0,Y 209.992,Z 802.5,A -85,B 0,C 180,E1 22987.331,E2 22987.331} C_VEL
LIN {X 0,Y 214.278,Z 787.002,A -85,B 0,C 180,E1 22989.912,E2 22989.912} C_VEL
LIN {X 0,Y 218.248,Z 770.814,A -85,B 0,C 180,E1 22991.98,E2 22991.98} C_VEL
LIN {X 0,Y 221.786,Z 753.675,A -85,B 0,C 180,E1 22993.612,E2 22993.612} C_VEL
LIN {X 0,Y 224.519,Z 735.763,A -85,B 0,C 180,E1 22994.81,E2 22994.81} C_VEL
LIN {X 0,Y 226.189,Z 717.5,A -85,B 0,C 180,E1 22995.611,E2 22995.611} C_VEL
LIN {X 0,Y 233.163,Z 583.947,A -85,B 0,C 180,E1 22999.406,E2 22999.406} C_VEL
LIN {X 0,Y 232.003,Z 565.156,A -85,B 0,C 180,E1 23000.37,E2 23000.37} C_VEL
LIN {X 0,Y 223.304,Z 547.979,A -85,B 0,C 180,E1 23002.89,E2 23002.89} C_VEL
LIN {X 0,Y 221.676,Z 544.687,A -85,B 0,C 180,E1 23003.461,E2 23003.461} C_VEL
LIN {X 0,Y 217.958,Z 532.367,A -85,B 0,C 180,E1 23007.851,E2 23007.851} C_VEL
LIN {X 0,Y 214.131,Z 521.193,A -85,B 0,C 180,E1 23012.522,E2 23012.522} C_VEL
LIN {X 0,Y 210.712,Z 512.125,A -85,B 0,C 180,E1 23017.009,E2 23017.009} C_VEL
LIN {X 0,Y 207.746,Z 504.936,A -85,B 0,C 180,E1 23021.189,E2 23021.189} C_VEL
LIN {X 0,Y 205.375,Z 499.842,A -85,B 0,C 180,E1 23024.758,E2 23024.758} C_VEL
LIN {X 0,Y 203.952,Z 496.613,A -85,B 0,C 180,E1 23027.256,E2 23027.256} C_VEL
LIN {X 0,Y 202.089,Z 492.536,A -85,B 0,C 180,E1 23030.891,E2 23030.891} C_VEL
LIN {X 0,Y 199.907,Z 488.079,A -85,B 0,C 180,E1 23035.985,E2 23035.985} C_VEL
LIN {X 0,Y 197.625,Z 483.498,A -85,B 0,C 180,E1 23044.062,E2 23044.062} C_VEL
LIN {X 0,Y 196.551,Z 482.186,A -85,B 0,C 180,E1 23050.553,E2 23050.553} C_VEL
LIN {X 0,Y 196.672,Z 482.351,A -85,B 0,C 180,E1 23057.102,E2 23057.102} C_VEL
LIN {X 0,Y 197.728,Z 483.795,A -85,B 0,C 180,E1 23062.916,E2 23062.916} C_VEL
LIN {X 0,Y 200,Z 488.52,A -85,B 0,C 180,E1 23070.993,E2 23070.993} C_VEL
LIN {X 0,Y 202.058,Z 493.198,A -85,B 0,C 180,E1 23076.235,E2 23076.235} C_VEL
LIN {X 0,Y 203.898,Z 497.485,A -85,B 0,C 180,E1 23080.094,E2 23080.094} C_VEL
LIN {X 0,Y 205.558,Z 501.625,A -85,B 0,C 180,E1 23083.303,E2 23083.303} C_VEL
LIN {X 0,Y 207.906,Z 507.467,A -85,B 0,C 180,E1 23087.304,E2 23087.304} C_VEL
LIN {X 0,Y 210.955,Z 516.215,A -85,B 0,C 180,E1 23092.329,E2 23092.329} C_VEL
LIN {X 0,Y 213.748,Z 525.403,A -85,B 0,C 180,E1 23096.859,E2 23096.859} C_VEL
LIN {X 0,Y 216.503,Z 535.808,A -85,B 0,C 180,E1 23101.339,E2 23101.339} C_VEL
LIN {X 0,Y 218.972,Z 547.313,A -85,B 0,C 180,E1 23105.735,E2 23105.735} C_VEL
LIN {X 0,Y 219.797,Z 551.048,A -85,B 0,C 180,E1 23106.95,E2 23106.95} C_VEL
LIN {X 0,Y 222.563,Z 557.394,A -85,B 0,C 180,E1 23107.854,E2 23107.854} C_VEL
LIN {X 0,Y 228.254,Z 608.226,A -85,B 0,C 180,E1 23111.125,E2 23111.125} C_VEL
LIN {X 0,Y 223.366,Z 693.474,A -85,B 0,C 180,E1 23113.774,E2 23113.774} C_VEL
LIN {X 0,Y 221.692,Z 710.888,A -85,B 0,C 180,E1 23114.798,E2 23114.798} C_VEL
LIN {X 0,Y 219.427,Z 726.467,A -85,B 0,C 180,E1 23116.159,E2 23116.159} C_VEL
LIN {X 0,Y 216.462,Z 741.808,A -85,B 0,C 180,E1 23118.003,E2 23118.003} C_VEL
LIN {X 0,Y 213.263,Z 755.449,A -85,B 0,C 180,E1 23120.146,E2 23120.146} C_VEL
LIN {X 0,Y 209.566,Z 769.023,A -85,B 0,C 180,E1 23122.932,E2 23122.932} C_VEL
LIN {X 0,Y 206.238,Z 780.116,A -85,B 0,C 180,E1 23125.829,E2 23125.829} C_VEL
LIN {X 0,Y 202.994,Z 790.236,A -85,B 0,C 180,E1 23129.193,E2 23129.193} C_VEL
LIN {X 0,Y 199.989,Z 799.475,A -85,B 0,C 180,E1 23133.152,E2 23133.152} C_VEL
LIN {X 0,Y 197.71,Z 806.77,A -85,B 0,C 180,E1 23137.263,E2 23137.263} C_VEL
LIN {X 0,Y 196.111,Z 812.628,A -85,B 0,C 180,E1 23141.788,E2 23141.788} C_VEL
LIN {X 0,Y 195.374,Z 816.702,A -85,B 0,C 180,E1 23146.348,E2 23146.348} C_VEL
LIN {X 0,Y 195.431,Z 819.091,A -85,B 0,C 180,E1 23150.985,E2 23150.985} C_VEL
LIN {X 0,Y 196.417,Z 819.888,A -85,B 0,C 180,E1 23155.962,E2 23155.962} C_VEL
LIN {X 0,Y 198.324,Z 818.964,A -85,B 0,C 180,E1 23160.61,E2 23160.61} C_VEL
LIN {X 0,Y 201.506,Z 816.033,A -85,B 0,C 180,E1 23165.488,E2 23165.488} C_VEL
LIN {X 0,Y 205.612,Z 811.412,A -85,B 0,C 180,E1 23169.933,E2 23169.933} C_VEL
LIN {X 0,Y 210.391,Z 805.165,A -85,B 0,C 180,E1 23173.935,E2 23173.935} C_VEL
LIN {X 0,Y 216.074,Z 796.877,A -85,B 0,C 180,E1 23177.763,E2 23177.763} C_VEL
LIN {X 0,Y 221.598,Z 787.698,A -85,B 0,C 180,E1 23180.901,E2 23180.901} C_VEL
LIN {X 0,Y 227.695,Z 776.168,A -85,B 0,C 180,E1 23183.899,E2 23183.899} C_VEL
LIN {X 0,Y 233.198,Z 764.125,A -85,B 0,C 180,E1 23186.283,E2 23186.283} C_VEL
LIN {X 0,Y 238.691,Z 749.729,A -85,B 0,C 180,E1 23188.455,E2 23188.455} C_VEL
LIN {X 0,Y 242.949,Z 736.075,A -85,B 0,C 180,E1 23190.033,E2 23190.033} C_VEL
LIN {X 0,Y 246.667,Z 720.503,A -85,B 0,C 180,E1 23191.375,E2 23191.375} C_VEL
LIN {X 0,Y 249.463,Z 703.927,A -85,B 0,C 180,E1 23192.393,E2 23192.393} C_VEL
LIN {X 0,Y 251.16,Z 686.297,A -85,B 0,C 180,E1 23193.07,E2 23193.07} C_VEL
LIN {X 0,Y 256.68,Z 615.794,A -85,B 0,C 180,E1 23195.013,E2 23195.013} C_VEL
LIN {X 0,Y 256.34,Z 611.493,A -85,B 0,C 180,E1 23195.367,E2 23195.367} C_VEL
LIN {X 0,Y 255.385,Z 605.593,A -85,B 0,C 180,E1 23196.039,E2 23196.039} C_VEL
LIN {X 0,Y 253.186,Z 598.793,A -85,B 0,C 180,E1 23197.259,E2 23197.259} C_VEL
LIN {X 0,Y 249.007,Z 590.162,A -85,B 0,C 180,E1 23199.513,E2 23199.513} C_VEL
LIN {X 0,Y 246.931,Z 586.123,A -85,B 0,C 180,E1 23200.72,E2 23200.72} C_VEL
LIN {X 0,Y 242.331,Z 577.102,A -85,B 0,C 180,E1 23203.705,E2 23203.705} C_VEL
LIN {X 0,Y 238.115,Z 569.819,A -85,B 0,C 180,E1 23206.894,E2 23206.894} C_VEL
LIN {X 0,Y 234.447,Z 563.643,A -85,B 0,C 180,E1 23210.301,E2 23210.301} C_VEL
LIN {X 0,Y 230.772,Z 557.802,A -85,B 0,C 180,E1 23214.904,E2 23214.904} C_VEL
LIN {X 0,Y 229.115,Z 555.106,A -85,B 0,C 180,E1 23217.935,E2 23217.935} C_VEL
LIN {X 0,Y 227.634,Z 552.197,A -85,B 0,C 180,E1 23224.282,E2 23224.282} C_VEL
LIN {X 0,Y 228.564,Z 552.727,A -85,B 0,C 180,E1 23230.179,E2 23230.179} C_VEL
LIN {X 0,Y 230.106,Z 554.503,A -85,B 0,C 180,E1 23233.57,E2 23233.57} C_VEL
LIN {X 0,Y 233.257,Z 558.393,A -85,B 0,C 180,E1 23237.976,E2 23237.976} C_VEL
LIN {X 0,Y 236.662,Z 562.751,A -85,B 0,C 180,E1 23241.37,E2 23241.37} C_VEL
LIN {X 0,Y 241.605,Z 569.818,A -85,B 0,C 180,E1 23245.295,E2 23245.295} C_VEL
LIN {X 0,Y 245.964,Z 576.507,A -85,B 0,C 180,E1 23248.134,E2 23248.134} C_VEL
LIN {X 0,Y 250.973,Z 584.857,A -85,B 0,C 180,E1 23250.992,E2 23250.992} C_VEL
LIN {X 0,Y 255.888,Z 594.126,A -85,B 0,C 180,E1 23253.471,E2 23253.471} C_VEL
LIN {X 0,Y 246.001,Z 719.835,A -85,B 0,C 180,E1 23256.715,E2 23256.715} C_VEL
LIN {X 0,Y 243.123,Z 737.883,A -85,B 0,C 180,E1 23257.466,E2 23257.466} C_VEL
LIN {X 0,Y 238.96,Z 755.327,A -85,B 0,C 180,E1 23258.516,E2 23258.516} C_VEL
LIN {X 0,Y 233.778,Z 771.936,A -85,B 0,C 180,E1 23259.907,E2 23259.907} C_VEL
LIN {X 0,Y 227.732,Z 787.807,A -85,B 0,C 180,E1 23261.722,E2 23261.722} C_VEL
LIN {X 0,Y 221.052,Z 802.865,A -85,B 0,C 180,E1 23264.013,E2 23264.013} C_VEL
LIN {X 0,Y 214.049,Z 816.88,A -85,B 0,C 180,E1 23266.818,E2 23266.818} C_VEL
LIN {X 0,Y 207.138,Z 829.539,A -85,B 0,C 180,E1 23270.129,E2 23270.129} C_VEL
LIN {X 0,Y 200.611,Z 840.765,A -85,B 0,C 180,E1 23273.977,E2 23273.977} C_VEL
LIN {X 0,Y 194.799,Z 850.656,A -85,B 0,C 180,E1 23278.433,E2 23278.433} C_VEL
LIN {X 0,Y 190.072,Z 859.054,A -85,B 0,C 180,E1 23283.441,E2 23283.441} C_VEL
LIN {X 0,Y 186.802,Z 865.937,A -85,B 0,C 180,E1 23288.985,E2 23288.985} C_VEL
LIN {X 0,Y 185.268,Z 870.882,A -85,B 0,C 180,E1 23294.667,E2 23294.667} C_VEL
LIN {X 0,Y 185.349,Z 873.978,A -85,B 0,C 180,E1 23300.374,E2 23300.374} C_VEL
LIN {X 0,Y 186.488,Z 875.255,A -85,B 0,C 180,E1 23305.736,E2 23305.736} C_VEL
LIN {X 0,Y 187.274,Z 875.072,A -85,B 0,C 180,E1 23309.389,E2 23309.389} C_VEL
LIN {X 0,Y 187.057,Z 874.008,A -85,B 0,C 180,E1 23312.758,E2 23312.758} C_VEL
LIN {X 0,Y 186.075,Z 871.079,A -85,B 0,C 180,E1 23317.41,E2 23317.41} C_VEL
LIN {X 0,Y 185.539,Z 866.303,A -85,B 0,C 180,E1 23322.449,E2 23322.449} C_VEL
LIN {X 0,Y 185.995,Z 859.739,A -85,B 0,C 180,E1 23327.521,E2 23327.521} C_VEL
LIN {X 0,Y 187.657,Z 851.156,A -85,B 0,C 180,E1 23332.559,E2 23332.559} C_VEL
LIN {X 0,Y 190.41,Z 841.055,A -85,B 0,C 180,E1 23337.184,E2 23337.184} C_VEL
LIN {X 0,Y 194.004,Z 829.47,A -85,B 0,C 180,E1 23341.369,E2 23341.369} C_VEL
LIN {X 0,Y 198.256,Z 816.378,A -85,B 0,C 180,E1 23345.096,E2 23345.096} C_VEL
LIN {X 0,Y 202.635,Z 802.42,A -85,B 0,C 180,E1 23348.203,E2 23348.203} C_VEL
LIN {X 0,Y 207.082,Z 787.056,A -85,B 0,C 180,E1 23350.862,E2 23350.862} C_VEL
LIN {X 0,Y 211.184,Z 771.08,A -85,B 0,C 180,E1 23352.983,E2 23352.983} C_VEL
LIN {X 0,Y 214.832,Z 754.237,A -85,B 0,C 180,E1 23354.651,E2 23354.651} C_VEL
LIN {X 0,Y 217.742,Z 736.453,A -85,B 0,C 180,E1 23355.908,E2 23355.908} C_VEL
LIN {X 0,Y 219.548,Z 718.169,A -85,B 0,C 180,E1 23356.752,E2 23356.752} C_VEL
LIN {X 0,Y 226.834,Z 584.682,A -85,B 0,C 180,E1 23360.621,E2 23360.621} C_VEL
LIN {X 0,Y 225.85,Z 568.202,A -85,B 0,C 180,E1 23361.497,E2 23361.497} C_VEL
LIN {X 0,Y 217.067,Z 550.764,A -85,B 0,C 180,E1 23364.198,E2 23364.198} C_VEL
LIN {X 0,Y 213.834,Z 544.552,A -85,B 0,C 180,E1 23365.382,E2 23365.382} C_VEL
LIN {X 0,Y 210.18,Z 532.601,A -85,B 0,C 180,E1 23370.033,E2 23370.033} C_VEL
LIN {X 0,Y 206.799,Z 522.815,A -85,B 0,C 180,E1 23374.513,E2 23374.513} C_VEL
LIN {X 0,Y 203.47,Z 513.962,A -85,B 0,C 180,E1 23379.28,E2 23379.28} C_VEL
LIN {X 0,Y 200.431,Z 506.663,A -85,B 0,C 180,E1 23384.076,E2 23384.076} C_VEL
LIN {X 0,Y 198.448,Z 502.366,A -85,B 0,C 180,E1 23387.488,E2 23387.488} C_VEL
LIN {X 0,Y 196.607,Z 498.295,A -85,B 0,C 180,E1 23391.225,E2 23391.225} C_VEL
LIN {X 0,Y 194.61,Z 494.051,A -85,B 0,C 180,E1 23396.171,E2 23396.171} C_VEL
LIN {X 0,Y 192.45,Z 489.59,A -85,B 0,C 180,E1 23404.172,E2 23404.172} C_VEL
LIN {X 0,Y 191.388,Z 488.297,A -85,B 0,C 180,E1 23410.841,E2 23410.841} C_VEL
LIN {X 0,Y 191.523,Z 488.488,A -85,B 0,C 180,E1 23417.312,E2 23417.312} C_VEL
LIN {X 0,Y 192.442,Z 489.722,A -85,B 0,C 180,E1 23422.612,E2 23422.612} C_VEL
LIN {X 0,Y 194.571,Z 494.467,A -85,B 0,C 180,E1 23430.923,E2 23430.923} C_VEL
LIN {X 0,Y 196.44,Z 498.843,A -85,B 0,C 180,E1 23435.972,E2 23435.972} C_VEL
LIN {X 0,Y 198.191,Z 503.127,A -85,B 0,C 180,E1 23439.929,E2 23439.929} C_VEL
LIN {X 0,Y 199.835,Z 507.349,A -85,B 0,C 180,E1 23443.273,E2 23443.273} C_VEL
LIN {X 0,Y 201.939,Z 512.861,A -85,B 0,C 180,E1 23447.122,E2 23447.122} C_VEL
LIN {X 0,Y 204.736,Z 521.151,A -85,B 0,C 180,E1 23452.023,E2 23452.023} C_VEL
LIN {X 0,Y 207.42,Z 530.323,A -85,B 0,C 180,E1 23456.664,E2 23456.664} C_VEL
LIN {X 0,Y 210.212,Z 541.578,A -85,B 0,C 180,E1 23461.598,E2 23461.598} C_VEL
LIN {X 0,Y 212.159,Z 550.818,A -85,B 0,C 180,E1 23465.105,E2 23465.105} C_VEL
LIN {X 0,Y 216.714,Z 560.811,A -85,B 0,C 180,E1 23466.677,E2 23466.677} C_VEL
LIN {X 0,Y 221.883,Z 609.366,A -85,B 0,C 180,E1 23469.903,E2 23469.903} C_VEL
LIN {X 0,Y 216.824,Z 694.09,A -85,B 0,C 180,E1 23472.583,E2 23472.583} C_VEL
LIN {X 0,Y 215.077,Z 711.508,A -85,B 0,C 180,E1 23473.629,E2 23473.629} C_VEL
LIN {X 0,Y 212.714,Z 727.106,A -85,B 0,C 180,E1 23475.017,E2 23475.017} C_VEL
LIN {X 0,Y 209.616,Z 742.482,A -85,B 0,C 180,E1 23476.904,E2 23476.904} C_VEL
LIN {X 0,Y 206.271,Z 756.164,A -85,B 0,C 180,E1 23479.102,E2 23479.102} C_VEL
LIN {X 0,Y 202.471,Z 769.534,A -85,B 0,C 180,E1 23481.909,E2 23481.909} C_VEL
LIN {X 0,Y 198.683,Z 781.607,A -85,B 0,C 180,E1 23485.161,E2 23485.161} C_VEL
LIN {X 0,Y 195.005,Z 792.489,A -85,B 0,C 180,E1 23488.991,E2 23488.991} C_VEL
LIN {X 0,Y 192.032,Z 801.263,A -85,B 0,C 180,E1 23492.984,E2 23492.984} C_VEL
LIN {X 0,Y 189.572,Z 808.8,A -85,B 0,C 180,E1 23497.576,E2 23497.576} C_VEL
LIN {X 0,Y 188.044,Z 814.426,A -85,B 0,C 180,E1 23502.279,E2 23502.279} C_VEL
LIN {X 0,Y 187.391,Z 818.361,A -85,B 0,C 180,E1 23507.235,E2 23507.235} C_VEL
LIN {X 0,Y 187.706,Z 820.651,A -85,B 0,C 180,E1 23512.552,E2 23512.552} C_VEL
LIN {X 0,Y 189.07,Z 820.997,A -85,B 0,C 180,E1 23517.734,E2 23517.734} C_VEL
LIN {X 0,Y 191.621,Z 819.493,A -85,B 0,C 180,E1 23522.864,E2 23522.864} C_VEL
LIN {X 0,Y 195.164,Z 816.267,A -85,B 0,C 180,E1 23527.564,E2 23527.564} C_VEL
LIN {X 0,Y 200.041,Z 810.878,A -85,B 0,C 180,E1 23532.289,E2 23532.289} C_VEL
LIN {X 0,Y 205.263,Z 804.29,A -85,B 0,C 180,E1 23536.234,E2 23536.234} C_VEL
LIN {X 0,Y 211.379,Z 795.498,A -85,B 0,C 180,E1 23540.021,E2 23540.021} C_VEL
LIN {X 0,Y 217.375,Z 785.786,A -85,B 0,C 180,E1 23543.163,E2 23543.163} C_VEL
LIN {X 0,Y 223.365,Z 774.598,A -85,B 0,C 180,E1 23545.906,E2 23545.906} C_VEL
LIN {X 0,Y 229.203,Z 761.954,A -85,B 0,C 180,E1 23548.282,E2 23548.282} C_VEL
LIN {X 0,Y 234.408,Z 748.475,A -85,B 0,C 180,E1 23550.229,E2 23550.229} C_VEL
LIN {X 0,Y 239.142,Z 733.027,A -85,B 0,C 180,E1 23551.908,E2 23551.908} C_VEL
LIN {X 0,Y 242.839,Z 717.134,A -85,B 0,C 180,E1 23553.181,E2 23553.181} C_VEL
LIN {X 0,Y 245.407,Z 700.518,A -85,B 0,C 180,E1 23554.095,E2 23554.095} C_VEL
LIN {X 0,Y 247.477,Z 676.967,A -85,B 0,C 180,E1 23554.875,E2 23554.875} C_VEL
LIN {X 0,Y 252.343,Z 617.39,A -85,B 0,C 180,E1 23556.502,E2 23556.502} C_VEL
LIN {X 0,Y 250.366,Z 593.315,A -85,B 0,C 180,E1 23558.72,E2 23558.72} C_VEL
LIN {X 0,Y 246.931,Z 586.123,A -85,B 0,C 180,E1 23560.72,E2 23560.72} C_VEL
LIN {X 0,Y 244.792,Z 582.938,A -85,B 0,C 180,E1 23561.983,E2 23561.983} C_VEL
LIN {X 0,Y 241.237,Z 580.138,A -85,B 0,C 180,E1 23564.096,E2 23564.096} C_VEL
LIN {X 0,Y 236.155,Z 576.695,A -85,B 0,C 180,E1 23567.613,E2 23567.613} C_VEL
LIN {X 0,Y 235.286,Z 575.533,A -85,B 0,C 180,E1 23568.359,E2 23568.359} C_VEL
LIN {X 0,Y 232.477,Z 570.624,A -85,B 0,C 180,E1 23571.217,E2 23571.217} C_VEL
LIN {X 0,Y 229.2,Z 565.059,A -85,B 0,C 180,E1 23575.746,E2 23575.746} C_VEL
LIN {X 0,Y 227.937,Z 562.932,A -85,B 0,C 180,E1 23578.24,E2 23578.24} C_VEL
LIN {X 0,Y 226.613,Z 560.129,A -85,B 0,C 180,E1 23584.33,E2 23584.33} C_VEL
LIN {X 0,Y 227.536,Z 560.669,A -85,B 0,C 180,E1 23590.161,E2 23590.161} C_VEL
LIN {X 0,Y 229.246,Z 562.736,A -85,B 0,C 180,E1 23593.879,E2 23593.879} C_VEL
LIN {X 0,Y 231.944,Z 566.277,A -85,B 0,C 180,E1 23597.697,E2 23597.697} C_VEL
LIN {X 0,Y 234.939,Z 570.24,A -85,B 0,C 180,E1 23600.815,E2 23600.815} C_VEL
LIN {X 0,Y 239.477,Z 576.986,A -85,B 0,C 180,E1 23604.612,E2 23604.612} C_VEL
LIN {X 0,Y 243.508,Z 583.408,A -85,B 0,C 180,E1 23607.379,E2 23607.379} C_VEL
LIN {X 0,Y 248.158,Z 591.465,A -85,B 0,C 180,E1 23610.174,E2 23610.174} C_VEL
LIN {X 0,Y 251.507,Z 598.213,A -85,B 0,C 180,E1 23612.011,E2 23612.011} C_VEL
LIN {X 0,Y 241.603,Z 719.252,A -85,B 0,C 180,E1 23615.133,E2 23615.133} C_VEL
LIN {X 0,Y 238.624,Z 737.285,A -85,B 0,C 180,E1 23615.879,E2 23615.879} C_VEL
LIN {X 0,Y 234.421,Z 754.361,A -85,B 0,C 180,E1 23616.896,E2 23616.896} C_VEL
LIN {X 0,Y 229.156,Z 770.717,A -85,B 0,C 180,E1 23618.245,E2 23618.245} C_VEL
LIN {X 0,Y 223.105,Z 786.114,A -85,B 0,C 180,E1 23619.974,E2 23619.974} C_VEL
LIN {X 0,Y 216.43,Z 800.64,A -85,B 0,C 180,E1 23622.143,E2 23622.143} C_VEL
LIN {X 0,Y 209.04,Z 814.811,A -85,B 0,C 180,E1 23624.936,E2 23624.936} C_VEL
LIN {X 0,Y 202.051,Z 827.031,A -85,B 0,C 180,E1 23628.084,E2 23628.084} C_VEL
LIN {X 0,Y 194.912,Z 838.685,A -85,B 0,C 180,E1 23632.007,E2 23632.007} C_VEL
LIN {X 0,Y 188.555,Z 848.751,A -85,B 0,C 180,E1 23636.532,E2 23636.532} C_VEL
LIN {X 0,Y 183.267,Z 857.29,A -85,B 0,C 180,E1 23641.664,E2 23641.664} C_VEL
LIN {X 0,Y 179.458,Z 864.276,A -85,B 0,C 180,E1 23647.392,E2 23647.392} C_VEL
LIN {X 0,Y 177.489,Z 869.353,A -85,B 0,C 180,E1 23653.304,E2 23653.304} C_VEL
LIN {X 0,Y 177.272,Z 872.603,A -85,B 0,C 180,E1 23659.274,E2 23659.274} C_VEL
LIN {X 0,Y 178.309,Z 874.008,A -85,B 0,C 180,E1 23664.853,E2 23664.853} C_VEL
LIN {X 0,Y 179.321,Z 873.882,A -85,B 0,C 180,E1 23669.042,E2 23669.042} C_VEL
LIN {X 0,Y 179.225,Z 872.961,A -85,B 0,C 180,E1 23672.239,E2 23672.239} C_VEL
LIN {X 0,Y 178.189,Z 870.136,A -85,B 0,C 180,E1 23677.092,E2 23677.092} C_VEL
LIN {X 0,Y 177.59,Z 865.455,A -85,B 0,C 180,E1 23682.354,E2 23682.354} C_VEL
LIN {X 0,Y 178.037,Z 858.991,A -85,B 0,C 180,E1 23687.654,E2 23687.654} C_VEL
LIN {X 0,Y 179.757,Z 850.535,A -85,B 0,C 180,E1 23692.915,E2 23692.915} C_VEL
LIN {X 0,Y 182.624,Z 840.532,A -85,B 0,C 180,E1 23697.735,E2 23697.735} C_VEL
LIN {X 0,Y 186.367,Z 829.05,A -85,B 0,C 180,E1 23702.083,E2 23702.083} C_VEL
LIN {X 0,Y 190.791,Z 816.072,A -85,B 0,C 180,E1 23705.941,E2 23705.941} C_VEL
LIN {X 0,Y 195.408,Z 802.067,A -85,B 0,C 180,E1 23709.193,E2 23709.193} C_VEL
LIN {X 0,Y 199.948,Z 787.068,A -85,B 0,C 180,E1 23711.881,E2 23711.881} C_VEL
LIN {X 0,Y 204.189,Z 771.259,A -85,B 0,C 180,E1 23714.055,E2 23714.055} C_VEL
LIN {X 0,Y 207.953,Z 754.654,A -85,B 0,C 180,E1 23715.759,E2 23715.759} C_VEL
LIN {X 0,Y 211.03,Z 736.867,A -85,B 0,C 180,E1 23717.069,E2 23717.069} C_VEL
LIN {X 0,Y 212.961,Z 718.784,A -85,B 0,C 180,E1 23717.95,E2 23717.95} C_VEL
LIN {X 0,Y 220.583,Z 585.467,A -85,B 0,C 180,E1 23721.891,E2 23721.891} C_VEL
LIN {X 0,Y 219.758,Z 571.263,A -85,B 0,C 180,E1 23722.681,E2 23722.681} C_VEL
LIN {X 0,Y 211.168,Z 554.111,A -85,B 0,C 180,E1 23725.5,E2 23725.5} C_VEL
LIN {X 0,Y 206.268,Z 545.131,A -85,B 0,C 180,E1 23727.284,E2 23727.284} C_VEL
LIN {X 0,Y 202.946,Z 534.332,A -85,B 0,C 180,E1 23731.774,E2 23731.774} C_VEL
LIN {X 0,Y 199.731,Z 525.002,A -85,B 0,C 180,E1 23736.392,E2 23736.392} C_VEL
LIN {X 0,Y 196.422,Z 516.198,A -85,B 0,C 180,E1 23741.603,E2 23741.603} C_VEL
LIN {X 0,Y 193.829,Z 510.281,A -85,B 0,C 180,E1 23745.97,E2 23745.97} C_VEL
LIN {X 0,Y 192.575,Z 507.516,A -85,B 0,C 180,E1 23748.318,E2 23748.318} C_VEL
LIN {X 0,Y 191.138,Z 504.056,A -85,B 0,C 180,E1 23751.578,E2 23751.578} C_VEL
LIN {X 0,Y 189.308,Z 500.017,A -85,B 0,C 180,E1 23756.367,E2 23756.367} C_VEL
LIN {X 0,Y 187.271,Z 495.68,A -85,B 0,C 180,E1 23764.287,E2 23764.287} C_VEL
LIN {X 0,Y 186.249,Z 494.427,A -85,B 0,C 180,E1 23770.831,E2 23770.831} C_VEL
LIN {X 0,Y 186.336,Z 494.574,A -85,B 0,C 180,E1 23777.227,E2 23777.227} C_VEL
LIN {X 0,Y 187.19,Z 495.811,A -85,B 0,C 180,E1 23782.619,E2 23782.619} C_VEL
LIN {X 0,Y 189.073,Z 500.115,A -85,B 0,C 180,E1 23790.51,E2 23790.51} C_VEL
LIN {X 0,Y 190.833,Z 504.495,A -85,B 0,C 180,E1 23795.696,E2 23795.696} C_VEL
LIN {X 0,Y 192.472,Z 508.709,A -85,B 0,C 180,E1 23799.716,E2 23799.716} C_VEL
LIN {X 0,Y 194.233,Z 513.343,A -85,B 0,C 180,E1 23803.461,E2 23803.461} C_VEL
LIN {X 0,Y 196.749,Z 520.393,A -85,B 0,C 180,E1 23808.336,E2 23808.336} C_VEL
LIN {X 0,Y 199.544,Z 529.576,A -85,B 0,C 180,E1 23813.592,E2 23813.592} C_VEL
LIN {X 0,Y 202.076,Z 539.321,A -85,B 0,C 180,E1 23818.366,E2 23818.366} C_VEL
LIN {X 0,Y 204.396,Z 549.994,A -85,B 0,C 180,E1 23822.913,E2 23822.913} C_VEL
LIN {X 0,Y 210.775,Z 563.498,A -85,B 0,C 180,E1 23825.356,E2 23825.356} C_VEL
LIN {X 0,Y 215.639,Z 609.834,A -85,B 0,C 180,E1 23828.597,E2 23828.597} C_VEL
LIN {X 0,Y 210.366,Z 694.575,A -85,B 0,C 180,E1 23831.323,E2 23831.323} C_VEL
LIN {X 0,Y 208.55,Z 711.959,A -85,B 0,C 180,E1 23832.383,E2 23832.383} C_VEL
LIN {X 0,Y 206.107,Z 727.524,A -85,B 0,C 180,E1 23833.788,E2 23833.788} C_VEL
LIN {X 0,Y 202.845,Z 743.069,A -85,B 0,C 180,E1 23835.731,E2 23835.731} C_VEL
LIN {X 0,Y 199.146,Z 757.512,A -85,B 0,C 180,E1 23838.12,E2 23838.12} C_VEL
LIN {X 0,Y 195.182,Z 770.806,A -85,B 0,C 180,E1 23841.011,E2 23841.011} C_VEL
LIN {X 0,Y 191.301,Z 782.601,A -85,B 0,C 180,E1 23844.3,E2 23844.3} C_VEL
LIN {X 0,Y 187.529,Z 793.252,A -85,B 0,C 180,E1 23848.166,E2 23848.166} C_VEL
LIN {X 0,Y 184.271,Z 802.42,A -85,B 0,C 180,E1 23852.487,E2 23852.487} C_VEL
LIN {X 0,Y 181.701,Z 809.949,A -85,B 0,C 180,E1 23857.27,E2 23857.27} C_VEL
LIN {X 0,Y 180.095,Z 815.672,A -85,B 0,C 180,E1 23862.274,E2 23862.274} C_VEL
LIN {X 0,Y 179.45,Z 819.609,A -85,B 0,C 180,E1 23867.51,E2 23867.51} C_VEL
LIN {X 0,Y 179.831,Z 821.826,A -85,B 0,C 180,E1 23872.904,E2 23872.904} C_VEL
LIN {X 0,Y 181.221,Z 822.235,A -85,B 0,C 180,E1 23878.019,E2 23878.019} C_VEL
LIN {X 0,Y 183.874,Z 820.862,A -85,B 0,C 180,E1 23883.312,E2 23883.312} C_VEL
LIN {X 0,Y 187.594,Z 817.826,A -85,B 0,C 180,E1 23888.189,E2 23888.189} C_VEL
LIN {X 0,Y 192.498,Z 812.811,A -85,B 0,C 180,E1 23892.913,E2 23892.913} C_VEL
LIN {X 0,Y 198.034,Z 806.368,A -85,B 0,C 180,E1 23897.062,E2 23897.062} C_VEL
LIN {X 0,Y 204.175,Z 798.24,A -85,B 0,C 180,E1 23900.822,E2 23900.822} C_VEL
LIN {X 0,Y 211.011,Z 787.861,A -85,B 0,C 180,E1 23904.35,E2 23904.35} C_VEL
LIN {X 0,Y 217.157,Z 777.181,A -85,B 0,C 180,E1 23907.09,E2 23907.09} C_VEL
LIN {X 0,Y 223.306,Z 764.66,A -85,B 0,C 180,E1 23909.533,E2 23909.533} C_VEL
LIN {X 0,Y 228.911,Z 751.056,A -85,B 0,C 180,E1 23911.568,E2 23911.568} C_VEL
LIN {X 0,Y 233.61,Z 737,A -85,B 0,C 180,E1 23913.174,E2 23913.174} C_VEL
LIN {X 0,Y 237.607,Z 721.346,A -85,B 0,C 180,E1 23914.504,E2 23914.504} C_VEL
LIN {X 0,Y 240.59,Z 704.828,A -85,B 0,C 180,E1 23915.503,E2 23915.503} C_VEL
LIN {X 0,Y 242.467,Z 686.428,A -85,B 0,C 180,E1 23916.196,E2 23916.196} C_VEL
LIN {X 0,Y 248.182,Z 618.991,A -85,B 0,C 180,E1 23918.042,E2 23918.042} C_VEL
LIN {X 0,Y 246.683,Z 598.138,A -85,B 0,C 180,E1 23920.032,E2 23920.032} C_VEL
LIN {X 0,Y 242.483,Z 589.003,A -85,B 0,C 180,E1 23922.729,E2 23922.729} C_VEL
LIN {X 0,Y 239,Z 582.349,A -85,B 0,C 180,E1 23925.214,E2 23925.214} C_VEL
LIN {X 0,Y 236.073,Z 576.906,A -85,B 0,C 180,E1 23927.649,E2 23927.649} C_VEL
LIN {X 0,Y 235.286,Z 575.533,A -85,B 0,C 180,E1 23928.359,E2 23928.359} C_VEL
LIN {X 0,Y 233.468,Z 573.674,A -85,B 0,C 180,E1 23930.001,E2 23930.001} C_VEL
LIN {X 0,Y 230.566,Z 573.117,A -85,B 0,C 180,E1 23932.81,E2 23932.81} C_VEL
LIN {X 0,Y 228.037,Z 572.682,A -85,B 0,C 180,E1 23935.992,E2 23935.992} C_VEL
LIN {X 0,Y 227.501,Z 571.959,A -85,B 0,C 180,E1 23936.956,E2 23936.956} C_VEL
LIN {X 0,Y 226.348,Z 570.146,A -85,B 0,C 180,E1 23939.746,E2 23939.746} C_VEL
LIN {X 0,Y 225.585,Z 568.044,A -85,B 0,C 180,E1 23944.575,E2 23944.575} C_VEL
LIN {X 0,Y 226.516,Z 568.619,A -85,B 0,C 180,E1 23950.169,E2 23950.169} C_VEL
LIN {X 0,Y 228.458,Z 571.142,A -85,B 0,C 180,E1 23954.316,E2 23954.316} C_VEL
LIN {X 0,Y 230.63,Z 574.141,A -85,B 0,C 180,E1 23957.405,E2 23957.405} C_VEL
LIN {X 0,Y 233.298,Z 577.832,A -85,B 0,C 180,E1 23960.312,E2 23960.312} C_VEL
LIN {X 0,Y 237.403,Z 584.154,A -85,B 0,C 180,E1 23963.914,E2 23963.914} C_VEL
LIN {X 0,Y 241.179,Z 590.459,A -85,B 0,C 180,E1 23966.665,E2 23966.665} C_VEL
LIN {X 0,Y 245.67,Z 598.635,A -85,B 0,C 180,E1 23969.502,E2 23969.502} C_VEL
LIN {X 0,Y 247.335,Z 602.186,A -85,B 0,C 180,E1 23970.493,E2 23970.493} C_VEL
LIN {X 0,Y 237.392,Z 718.684,A -85,B 0,C 180,E1 23973.495,E2 23973.495} C_VEL
LIN {X 0,Y 234.291,Z 736.798,A -85,B 0,C 180,E1 23974.238,E2 23974.238} C_VEL
LIN {X 0,Y 230.077,Z 753.395,A -85,B 0,C 180,E1 23975.215,E2 23975.215} C_VEL
LIN {X 0,Y 224.637,Z 769.78,A -85,B 0,C 180,E1 23976.544,E2 23976.544} C_VEL
LIN {X 0,Y 218.361,Z 785.186,A -85,B 0,C 180,E1 23978.253,E2 23978.253} C_VEL
LIN {X 0,Y 211.093,Z 800.323,A -85,B 0,C 180,E1 23980.517,E2 23980.517} C_VEL
LIN {X 0,Y 203.389,Z 814.38,A -85,B 0,C 180,E1 23983.318,E2 23983.318} C_VEL
LIN {X 0,Y 196.064,Z 826.463,A -85,B 0,C 180,E1 23986.493,E2 23986.493} C_VEL
LIN {X 0,Y 188.528,Z 837.98,A -85,B 0,C 180,E1 23990.475,E2 23990.475} C_VEL
LIN {X 0,Y 181.76,Z 847.946,A -85,B 0,C 180,E1 23995.104,E2 23995.104} C_VEL
LIN {X 0,Y 176.069,Z 856.409,A -85,B 0,C 180,E1 24000.393,E2 24000.393} C_VEL
LIN {X 0,Y 171.891,Z 863.318,A -85,B 0,C 180,E1 24006.337,E2 24006.337} C_VEL
LIN {X 0,Y 169.65,Z 868.305,A -85,B 0,C 180,E1 24012.508,E2 24012.508} C_VEL
LIN {X 0,Y 169.31,Z 871.561,A -85,B 0,C 180,E1 24019.108,E2 24019.108} C_VEL
LIN {X 0,Y 170.393,Z 872.805,A -85,B 0,C 180,E1 24024.951,E2 24024.951} C_VEL
LIN {X 0,Y 171.403,Z 872.641,A -85,B 0,C 180,E1 24028.998,E2 24028.998} C_VEL
LIN {X 0,Y 171.341,Z 871.792,A -85,B 0,C 180,E1 24032.007,E2 24032.007} C_VEL
LIN {X 0,Y 170.242,Z 868.965,A -85,B 0,C 180,E1 24037.085,E2 24037.085} C_VEL
LIN {X 0,Y 169.627,Z 864.271,A -85,B 0,C 180,E1 24042.598,E2 24042.598} C_VEL
LIN {X 0,Y 170.152,Z 857.79,A -85,B 0,C 180,E1 24048.147,E2 24048.147} C_VEL
LIN {X 0,Y 172.025,Z 849.297,A -85,B 0,C 180,E1 24053.644,E2 24053.644} C_VEL
LIN {X 0,Y 175.103,Z 839.246,A -85,B 0,C 180,E1 24058.663,E2 24058.663} C_VEL
LIN {X 0,Y 179.084,Z 827.691,A -85,B 0,C 180,E1 24063.173,E2 24063.173} C_VEL
LIN {X 0,Y 183.764,Z 814.618,A -85,B 0,C 180,E1 24067.154,E2 24067.154} C_VEL
LIN {X 0,Y 188.621,Z 800.438,A -85,B 0,C 180,E1 24070.494,E2 24070.494} C_VEL
LIN {X 0,Y 193.379,Z 785.282,A -85,B 0,C 180,E1 24073.243,E2 24073.243} C_VEL
LIN {X 0,Y 197.814,Z 769.255,A -85,B 0,C 180,E1 24075.455,E2 24075.455} C_VEL
LIN {X 0,Y 201.729,Z 752.311,A -85,B 0,C 180,E1 24077.186,E2 24077.186} C_VEL
LIN {X 0,Y 204.764,Z 734.704,A -85,B 0,C 180,E1 24078.459,E2 24078.459} C_VEL
LIN {X 0,Y 206.667,Z 716.523,A -85,B 0,C 180,E1 24079.321,E2 24079.321} C_VEL
LIN {X 0,Y 214.447,Z 586.261,A -85,B 0,C 180,E1 24083.234,E2 24083.234} C_VEL
LIN {X 0,Y 213.838,Z 574.549,A -85,B 0,C 180,E1 24083.904,E2 24083.904} C_VEL
LIN {X 0,Y 205.908,Z 558.508,A -85,B 0,C 180,E1 24086.68,E2 24086.68} C_VEL
LIN {X 0,Y 198.696,Z 545.465,A -85,B 0,C 180,E1 24089.454,E2 24089.454} C_VEL
LIN {X 0,Y 195.374,Z 534.948,A -85,B 0,C 180,E1 24094.253,E2 24094.253} C_VEL
LIN {X 0,Y 192.535,Z 526.852,A -85,B 0,C 180,E1 24098.684,E2 24098.684} C_VEL
LIN {X 0,Y 190.062,Z 520.412,A -85,B 0,C 180,E1 24102.867,E2 24102.867} C_VEL
LIN {X 0,Y 187.709,Z 514.286,A -85,B 0,C 180,E1 24107.542,E2 24107.542} C_VEL
LIN {X 0,Y 185.513,Z 509.565,A -85,B 0,C 180,E1 24112.257,E2 24112.257} C_VEL
LIN {X 0,Y 184.007,Z 505.983,A -85,B 0,C 180,E1 24116.574,E2 24116.574} C_VEL
LIN {X 0,Y 182.089,Z 501.768,A -85,B 0,C 180,E1 24124.41,E2 24124.41} C_VEL
LIN {X 0,Y 181.079,Z 500.533,A -85,B 0,C 180,E1 24131.144,E2 24131.144} C_VEL
LIN {X 0,Y 181.198,Z 500.73,A -85,B 0,C 180,E1 24137.668,E2 24137.668} C_VEL
LIN {X 0,Y 181.941,Z 501.903,A -85,B 0,C 180,E1 24142.625,E2 24142.625} C_VEL
LIN {X 0,Y 183.657,Z 506.072,A -85,B 0,C 180,E1 24150.419,E2 24150.419} C_VEL
LIN {X 0,Y 185.234,Z 510.147,A -85,B 0,C 180,E1 24155.405,E2 24155.405} C_VEL
LIN {X 0,Y 186.683,Z 513.97,A -85,B 0,C 180,E1 24159.199,E2 24159.199} C_VEL
LIN {X 0,Y 188.814,Z 519.648,A -85,B 0,C 180,E1 24163.929,E2 24163.929} C_VEL
LIN {X 0,Y 191.507,Z 528.17,A -85,B 0,C 180,E1 24169.666,E2 24169.666} C_VEL
LIN {X 0,Y 194.033,Z 537.245,A -85,B 0,C 180,E1 24174.75,E2 24174.75} C_VEL
LIN {X 0,Y 196.405,Z 547.612,A -85,B 0,C 180,E1 24179.735,E2 24179.735} C_VEL
LIN {X 0,Y 197.215,Z 550.726,A -85,B 0,C 180,E1 24180.92,E2 24180.92} C_VEL
LIN {X 0,Y 204.739,Z 566.051,A -85,B 0,C 180,E1 24183.894,E2 24183.894} C_VEL
LIN {X 0,Y 205.382,Z 568.409,A -85,B 0,C 180,E1 24184.183,E2 24184.183} C_VEL
LIN {X 0,Y 209.426,Z 611.647,A -85,B 0,C 180,E1 24187.254,E2 24187.254} C_VEL
LIN {X 0,Y 204.003,Z 695.214,A -85,B 0,C 180,E1 24189.991,E2 24189.991} C_VEL
LIN {X 0,Y 202.087,Z 712.716,A -85,B 0,C 180,E1 24191.081,E2 24191.081} C_VEL
LIN {X 0,Y 199.553,Z 728.17,A -85,B 0,C 180,E1 24192.504,E2 24192.504} C_VEL
LIN {X 0,Y 196.079,Z 744.014,A -85,B 0,C 180,E1 24194.531,E2 24194.531} C_VEL
LIN {X 0,Y 192.327,Z 758.053,A -85,B 0,C 180,E1 24196.905,E2 24196.905} C_VEL
LIN {X 0,Y 188.133,Z 771.506,A -85,B 0,C 180,E1 24199.899,E2 24199.899} C_VEL
LIN {X 0,Y 184.217,Z 782.875,A -85,B 0,C 180,E1 24203.142,E2 24203.142} C_VEL
LIN {X 0,Y 180.501,Z 792.959,A -85,B 0,C 180,E1 24206.824,E2 24206.824} C_VEL
LIN {X 0,Y 176.957,Z 802.375,A -85,B 0,C 180,E1 24211.294,E2 24211.294} C_VEL
LIN {X 0,Y 174.296,Z 809.782,A -85,B 0,C 180,E1 24215.926,E2 24215.926} C_VEL
LIN {X 0,Y 172.432,Z 815.724,A -85,B 0,C 180,E1 24221.031,E2 24221.031} C_VEL
LIN {X 0,Y 171.56,Z 820.173,A -85,B 0,C 180,E1 24226.593,E2 24226.593} C_VEL
LIN {X 0,Y 171.792,Z 822.708,A -85,B 0,C 180,E1 24232.228,E2 24232.228} C_VEL
LIN {X 0,Y 173.245,Z 823.474,A -85,B 0,C 180,E1 24237.99,E2 24237.99} C_VEL
LIN {X 0,Y 175.925,Z 822.368,A -85,B 0,C 180,E1 24243.455,E2 24243.455} C_VEL
LIN {X 0,Y 180.042,Z 819.342,A -85,B 0,C 180,E1 24248.868,E2 24248.868} C_VEL
LIN {X 0,Y 185.151,Z 814.597,A -85,B 0,C 180,E1 24253.727,E2 24253.727} C_VEL
LIN {X 0,Y 191.417,Z 807.781,A -85,B 0,C 180,E1 24258.326,E2 24258.326} C_VEL
LIN {X 0,Y 197.726,Z 799.973,A -85,B 0,C 180,E1 24262.078,E2 24262.078} C_VEL
LIN {X 0,Y 204.753,Z 789.918,A -85,B 0,C 180,E1 24265.615,E2 24265.615} C_VEL
LIN {X 0,Y 211.544,Z 778.776,A -85,B 0,C 180,E1 24268.553,E2 24268.553} C_VEL
LIN {X 0,Y 217.921,Z 766.496,A -85,B 0,C 180,E1 24270.999,E2 24270.999} C_VEL
LIN {X 0,Y 224.108,Z 752.179,A -85,B 0,C 180,E1 24273.163,E2 24273.163} C_VEL
LIN {X 0,Y 229.22,Z 737.449,A -85,B 0,C 180,E1 24274.838,E2 24274.838} C_VEL
LIN {X 0,Y 233.378,Z 721.729,A -85,B 0,C 180,E1 24276.162,E2 24276.162} C_VEL
LIN {X 0,Y 236.46,Z 705.226,A -85,B 0,C 180,E1 24277.149,E2 24277.149} C_VEL
LIN {X 0,Y 238.44,Z 686.42,A -85,B 0,C 180,E1 24277.848,E2 24277.848} C_VEL
LIN {X 0,Y 244.253,Z 620.459,A -85,B 0,C 180,E1 24279.653,E2 24279.653} C_VEL
LIN {X 0,Y 243.14,Z 602.928,A -85,B 0,C 180,E1 24281.384,E2 24281.384} C_VEL
LIN {X 0,Y 239.218,Z 594.245,A -85,B 0,C 180,E1 24284.111,E2 24284.111} C_VEL
LIN {X 0,Y 236.585,Z 588.886,A -85,B 0,C 180,E1 24286.185,E2 24286.185} C_VEL
LIN {X 0,Y 233.946,Z 583.766,A -85,B 0,C 180,E1 24288.536,E2 24288.536} C_VEL
LIN {X 0,Y 230.99,Z 578.295,A -85,B 0,C 180,E1 24291.662,E2 24291.662} C_VEL
LIN {X 0,Y 227.873,Z 572.713,A -85,B 0,C 180,E1 24296.226,E2 24296.226} C_VEL
LIN {X 0,Y 227.501,Z 571.959,A -85,B 0,C 180,E1 24296.956,E2 24296.956} C_VEL
LIN {X 0,Y 226.626,Z 571.288,A -85,B 0,C 180,E1 24298.745,E2 24298.745} C_VEL
LIN {X 0,Y 225.523,Z 572.71,A -85,B 0,C 180,E1 24301.249,E2 24301.249} C_VEL
LIN {X 0,Y 224.593,Z 575.744,A -85,B 0,C 180,E1 24305.072,E2 24305.072} C_VEL
LIN {X 0,Y 224.605,Z 575.941,A -85,B 0,C 180,E1 24305.938,E2 24305.938} C_VEL
LIN {X 0,Y 225.781,Z 576.873,A -85,B 0,C 180,E1 24310.977,E2 24310.977} C_VEL
LIN {X 0,Y 228.7,Z 580.905,A -85,B 0,C 180,E1 24316.248,E2 24316.248} C_VEL
LIN {X 0,Y 231.624,Z 585.329,A -85,B 0,C 180,E1 24319.749,E2 24319.749} C_VEL
LIN {X 0,Y 235.434,Z 591.452,A -85,B 0,C 180,E1 24323.263,E2 24323.263} C_VEL
LIN {X 0,Y 238.969,Z 597.657,A -85,B 0,C 180,E1 24325.994,E2 24325.994} C_VEL
LIN {X 0,Y 243.326,Z 606.007,A -85,B 0,C 180,E1 24328.883,E2 24328.883} C_VEL
LIN {X 0,Y 233.437,Z 717.935,A -85,B 0,C 180,E1 24331.789,E2 24331.789} C_VEL
LIN {X 0,Y 230.255,Z 735.932,A -85,B 0,C 180,E1 24332.517,E2 24332.517} C_VEL
LIN {X 0,Y 225.94,Z 752.429,A -85,B 0,C 180,E1 24333.471,E2 24333.471} C_VEL
LIN {X 0,Y 220.327,Z 768.843,A -85,B 0,C 180,E1 24334.776,E2 24334.776} C_VEL
LIN {X 0,Y 213.826,Z 784.258,A -85,B 0,C 180,E1 24336.46,E2 24336.46} C_VEL
LIN {X 0,Y 206.269,Z 799.389,A -85,B 0,C 180,E1 24338.701,E2 24338.701} C_VEL
LIN {X 0,Y 198.361,Z 813.199,A -85,B 0,C 180,E1 24341.438,E2 24341.438} C_VEL
LIN {X 0,Y 190.24,Z 825.932,A -85,B 0,C 180,E1 24344.804,E2 24344.804} C_VEL
LIN {X 0,Y 182.292,Z 837.304,A -85,B 0,C 180,E1 24348.839,E2 24348.839} C_VEL
LIN {X 0,Y 175.089,Z 847.153,A -85,B 0,C 180,E1 24353.567,E2 24353.567} C_VEL
LIN {X 0,Y 168.811,Z 855.751,A -85,B 0,C 180,E1 24359.184,E2 24359.184} C_VEL
LIN {X 0,Y 164.387,Z 862.361,A -85,B 0,C 180,E1 24365.186,E2 24365.186} C_VEL
LIN {X 0,Y 161.844,Z 867.235,A -85,B 0,C 180,E1 24371.635,E2 24371.635} C_VEL
LIN {X 0,Y 161.303,Z 870.344,A -85,B 0,C 180,E1 24378.343,E2 24378.343} C_VEL
LIN {X 0,Y 162.383,Z 871.585,A -85,B 0,C 180,E1 24384.701,E2 24384.701} C_VEL
LIN {X 0,Y 163.538,Z 871.35,A -85,B 0,C 180,E1 24389.3,E2 24389.3} C_VEL
LIN {X 0,Y 163.32,Z 870.349,A -85,B 0,C 180,E1 24392.457,E2 24392.457} C_VEL
LIN {X 0,Y 162.161,Z 867.329,A -85,B 0,C 180,E1 24397.797,E2 24397.797} C_VEL
LIN {X 0,Y 161.675,Z 862.114,A -85,B 0,C 180,E1 24403.847,E2 24403.847} C_VEL
LIN {X 0,Y 162.552,Z 855.094,A -85,B 0,C 180,E1 24409.774,E2 24409.774} C_VEL
LIN {X 0,Y 164.877,Z 846.16,A -85,B 0,C 180,E1 24415.504,E2 24415.504} C_VEL
LIN {X 0,Y 168.447,Z 835.658,A -85,B 0,C 180,E1 24420.696,E2 24420.696} C_VEL
LIN {X 0,Y 172.719,Z 824.056,A -85,B 0,C 180,E1 24425.139,E2 24425.139} C_VEL
LIN {X 0,Y 177.673,Z 810.806,A -85,B 0,C 180,E1 24429.072,E2 24429.072} C_VEL
LIN {X 0,Y 182.768,Z 796.356,A -85,B 0,C 180,E1 24432.394,E2 24432.394} C_VEL
LIN {X 0,Y 187.72,Z 780.94,A -85,B 0,C 180,E1 24435.106,E2 24435.106} C_VEL
LIN {X 0,Y 192.132,Z 765.094,A -85,B 0,C 180,E1 24437.204,E2 24437.204} C_VEL
LIN {X 0,Y 195.967,Z 748.17,A -85,B 0,C 180,E1 24438.839,E2 24438.839} C_VEL
LIN {X 0,Y 198.948,Z 729.931,A -85,B 0,C 180,E1 24440.077,E2 24440.077} C_VEL
LIN {X 0,Y 200.685,Z 711.706,A -85,B 0,C 180,E1 24440.867,E2 24440.867} C_VEL
LIN {X 0,Y 208.434,Z 586.997,A -85,B 0,C 180,E1 24444.659,E2 24444.659} C_VEL
LIN {X 0,Y 207.949,Z 577.604,A -85,B 0,C 180,E1 24445.224,E2 24445.224} C_VEL
LIN {X 0,Y 199.585,Z 560.644,A -85,B 0,C 180,E1 24448.348,E2 24448.348} C_VEL
LIN {X 0,Y 191.16,Z 545.854,A -85,B 0,C 180,E1 24451.854,E2 24451.854} C_VEL
LIN {X 0,Y 188.323,Z 537.059,A -85,B 0,C 180,E1 24456.203,E2 24456.203} C_VEL
LIN {X 0,Y 185.677,Z 529.318,A -85,B 0,C 180,E1 24460.824,E2 24460.824} C_VEL
LIN {X 0,Y 183.061,Z 522.532,A -85,B 0,C 180,E1 24465.772,E2 24465.772} C_VEL
LIN {X 0,Y 181.578,Z 518.988,A -85,B 0,C 180,E1 24468.889,E2 24468.889} C_VEL
LIN {X 0,Y 180.198,Z 515.547,A -85,B 0,C 180,E1 24472.348,E2 24472.348} C_VEL
LIN {X 0,Y 178.573,Z 511.778,A -85,B 0,C 180,E1 24477.112,E2 24477.112} C_VEL
LIN {X 0,Y 176.904,Z 507.853,A -85,B 0,C 180,E1 24484.539,E2 24484.539} C_VEL
LIN {X 0,Y 175.929,Z 506.655,A -85,B 0,C 180,E1 24491.142,E2 24491.142} C_VEL
LIN {X 0,Y 176.044,Z 506.856,A -85,B 0,C 180,E1 24497.861,E2 24497.861} C_VEL
LIN {X 0,Y 176.697,Z 508.036,A -85,B 0,C 180,E1 24502.726,E2 24502.726} C_VEL
LIN {X 0,Y 178.249,Z 512.034,A -85,B 0,C 180,E1 24510.322,E2 24510.322} C_VEL
LIN {X 0,Y 179.658,Z 515.82,A -85,B 0,C 180,E1 24515.103,E2 24515.103} C_VEL
LIN {X 0,Y 181.023,Z 519.666,A -85,B 0,C 180,E1 24519.026,E2 24519.026} C_VEL
LIN {X 0,Y 183.008,Z 525.339,A -85,B 0,C 180,E1 24523.847,E2 24523.847} C_VEL
LIN {X 0,Y 185.367,Z 533.134,A -85,B 0,C 180,E1 24529.256,E2 24529.256} C_VEL
LIN {X 0,Y 187.657,Z 541.835,A -85,B 0,C 180,E1 24534.288,E2 24534.288} C_VEL
LIN {X 0,Y 189.634,Z 550.3,A -85,B 0,C 180,E1 24538.397,E2 24538.397} C_VEL
LIN {X 0,Y 196.181,Z 563.23,A -85,B 0,C 180,E1 24541.286,E2 24541.286} C_VEL
LIN {X 0,Y 199.753,Z 571.197,A -85,B 0,C 180,E1 24542.762,E2 24542.762} C_VEL
LIN {X 0,Y 203.384,Z 612.727,A -85,B 0,C 180,E1 24545.807,E2 24545.807} C_VEL
LIN {X 0,Y 197.758,Z 695.852,A -85,B 0,C 180,E1 24548.574,E2 24548.574} C_VEL
LIN {X 0,Y 195.751,Z 713.365,A -85,B 0,C 180,E1 24549.685,E2 24549.685} C_VEL
LIN {X 0,Y 193.13,Z 728.698,A -85,B 0,C 180,E1 24551.12,E2 24551.12} C_VEL
LIN {X 0,Y 189.585,Z 744.239,A -85,B 0,C 180,E1 24553.138,E2 24553.138} C_VEL
LIN {X 0,Y 185.53,Z 758.812,A -85,B 0,C 180,E1 24555.646,E2 24555.646} C_VEL
LIN {X 0,Y 181.161,Z 772.203,A -85,B 0,C 180,E1 24558.7,E2 24558.7} C_VEL
LIN {X 0,Y 176.864,Z 784.098,A -85,B 0,C 180,E1 24562.202,E2 24562.202} C_VEL
LIN {X 0,Y 172.967,Z 794.135,A -85,B 0,C 180,E1 24566.022,E2 24566.022} C_VEL
LIN {X 0,Y 169.25,Z 803.534,A -85,B 0,C 180,E1 24570.676,E2 24570.676} C_VEL
LIN {X 0,Y 166.459,Z 810.93,A -85,B 0,C 180,E1 24575.514,E2 24575.514} C_VEL
LIN {X 0,Y 164.512,Z 816.87,A -85,B 0,C 180,E1 24580.859,E2 24580.859} C_VEL
LIN {X 0,Y 163.622,Z 821.327,A -85,B 0,C 180,E1 24586.69,E2 24586.69} C_VEL
